(* CoDeSys 2.3 project: cy-wg-03_102.pro *)
(* Title: cy-003-wg (SanFelice) *)
(* Author: Andrea Ravasio *)
(* Libraries: serial_interface_01.lib 22.4.13 12:50:14, SerComm.lib 31.5.11 09:06:48, MBus_03.lib 9.2.13 17:51:58, Util.lib 26.9.14 11:12:46, Visual.lib 8.11.10 12:37:48, WagoLibIdent.lib 25.2.13 13:49:34, WagoLibStatus.lib 8.11.10 12:37:48, SysLibFile.lib 8.11.10 12:37:48, SysLibRtc.lib 8.11.10 12:37:48, SysLibSockets.lib 5.5.11 09:22:24, SysLibEvent.lib 8.11.10 12:37:48, SysLibPlcCtrl.lib 8.11.10 12:37:48, Standard.lib 8.11.10 12:37:48, SYSLIBCALLBACK.LIB 8.11.10 12:37:48, WagoLibDaylightSaving.lib 8.11.10 12:37:48, SysLibTime.lib 8.11.10 12:37:48, 32_Bit\DaylightSaving.lib 2.12.10 14:48:32 *)

(* PLC configuration (modules and I/O channels)
VPN_ST2 AT %IX16.0 [BOOLOnX_I] Ch_1 Digital input
KEY_QE_ST AT %IX16.1 [BOOLOnX_I] Ch_2 Digital input
SCA01_5_DI AT %IX16.2 [BOOLOnX_I] Ch_3 Digital input
PORT01_DI AT %IX16.3 [BOOLOnX_I] Ch_4 Digital input
0750-0402 4 DI 24 V DC 3.0ms [Type_1_4_Channels] node 1, in %IB32 out %QB8 {INTTypePAAssignment = PLC; INTTypeModule = plugged}
  GAS02_DI AT %IX16.4 [BOOLOnX_I] Ch_1 Digital input
  GAS01_DI AT %IX16.5 [BOOLOnX_I] Ch_2 Digital input
  SCA01_6_DI AT %IX16.6 [BOOLOnX_I] Ch_3 Digital input
  SCA05_1_DI AT %IX16.7 [BOOLOnX_I] Ch_4 Digital input
SCA05_2_DI AT %IX16.8 [BOOLOnX_I] Ch_1 Digital input
SCA01_1_DO AT %QX4.0 [BOOLOnX_Q] Ch_1 Digital output
SCA05_3_DI AT %IX16.9 [BOOLOnX_I] Ch_2 Digital input
SCA01_2_DO AT %QX4.1 [BOOLOnX_Q] Ch_2 Digital output
SCA05_4_DI AT %IX16.10 [BOOLOnX_I] Ch_3 Digital input
SCA01_3_DO AT %QX4.2 [BOOLOnX_Q] Ch_3 Digital output
SCA05_5_DI AT %IX16.11 [BOOLOnX_I] Ch_4 Digital input
SCA01_4_DO AT %QX4.3 [BOOLOnX_Q] Ch_4 Digital output
SCA05_6_DI AT %IX16.12 [BOOLOnX_I] Ch_5 Digital input
LAMP_AL AT %QX4.4 [BOOLOnX_Q] Ch_5 Digital output
AT %IX16.13 [BOOLOnX_I] Ch_6 Digital input
CAL02_RESET AT %QX4.5 [BOOLOnX_Q] Ch_6 Digital output
AT %IX16.14 [BOOLOnX_I] Ch_7 Digital input
CAL03_RESET AT %QX4.6 [BOOLOnX_Q] Ch_7 Digital output
SCA05_10_DI AT %IX16.15 [BOOLOnX_I] Ch_8 Digital input
AT %QX4.7 [BOOLOnX_Q] Ch_8 Digital output
SCA06_1_DI AT %IX17.0 [BOOLOnX_I] Ch_1 Digital input
CIRD02B_EN AT %QX4.8 [BOOLOnX_Q] Ch_1 Digital output
SCA06_2_DI AT %IX17.1 [BOOLOnX_I] Ch_2 Digital input
CIRD02A_EN AT %QX4.9 [BOOLOnX_Q] Ch_2 Digital output
SCA06_5_DI AT %IX17.2 [BOOLOnX_I] Ch_3 Digital input
CIRD01B_EN AT %QX4.10 [BOOLOnX_Q] Ch_3 Digital output
SCA06_6_DI AT %IX17.3 [BOOLOnX_I] Ch_4 Digital input
CIRD01A_EN AT %QX4.11 [BOOLOnX_Q] Ch_4 Digital output
SCA06_7_DI AT %IX17.4 [BOOLOnX_I] Ch_5 Digital input
EV02_EN AT %QX4.12 [BOOLOnX_Q] Ch_5 Digital output
SCA06_8_DI AT %IX17.5 [BOOLOnX_I] Ch_6 Digital input
EV03_EN AT %QX4.13 [BOOLOnX_Q] Ch_6 Digital output
SCA06_15_DI AT %IX17.6 [BOOLOnX_I] Ch_7 Digital input
CAL02_EN AT %QX4.14 [BOOLOnX_Q] Ch_7 Digital output
SCA06_16_DI AT %IX17.7 [BOOLOnX_I] Ch_8 Digital input
CAL03_EN AT %QX4.15 [BOOLOnX_Q] Ch_8 Digital output
0750-1506 8DI / 8DO 24V DC 0.5A [Type_34_8_Channels] node 4, in %IB34 out %QB9 {INTTypePAAssignment = PLC; INTTypeModule = plugged}
  SCA06_9_DI AT %IX17.8 [BOOLOnX_I] Ch_1 Digital input
  AT %QX5.0 [BOOLOnX_Q] Ch_1 Digital output
  SCA06_10_DI AT %IX17.9 [BOOLOnX_I] Ch_2 Digital input
  AT %QX5.1 [BOOLOnX_Q] Ch_2 Digital output
  SCA06_11_DI AT %IX17.10 [BOOLOnX_I] Ch_3 Digital input
  AT %QX5.2 [BOOLOnX_Q] Ch_3 Digital output
  SCA06_12_DI AT %IX17.11 [BOOLOnX_I] Ch_4 Digital input
  AT %QX5.3 [BOOLOnX_Q] Ch_4 Digital output
  SCA06_19_DI AT %IX17.12 [BOOLOnX_I] Ch_5 Digital input
  AT %QX5.4 [BOOLOnX_Q] Ch_5 Digital output
  SCA06_20_DI AT %IX17.13 [BOOLOnX_I] Ch_6 Digital input
  AT %QX5.5 [BOOLOnX_Q] Ch_6 Digital output
  CIRD01A_ST AT %IX17.14 [BOOLOnX_I] Ch_7 Digital input
  AT %QX5.6 [BOOLOnX_Q] Ch_7 Digital output
  CIRD01A_AL AT %IX17.15 [BOOLOnX_I] Ch_8 Digital input
  AT %QX5.7 [BOOLOnX_Q] Ch_8 Digital output
0750-1506 8DI / 8DO 24V DC 0.5A [Type_34_8_Channels] node 5, in %IB35 out %QB10 {INTTypePAAssignment = PLC; INTTypeModule = plugged}
  CIRD01B_ST AT %IX18.0 [BOOLOnX_I] Ch_1 Digital input
  AT %QX5.8 [BOOLOnX_Q] Ch_1 Digital output
  CIRD01B_AL AT %IX18.1 [BOOLOnX_I] Ch_2 Digital input
  AT %QX5.9 [BOOLOnX_Q] Ch_2 Digital output
  CIRD02A_ST AT %IX18.2 [BOOLOnX_I] Ch_3 Digital input
  AT %QX5.10 [BOOLOnX_Q] Ch_3 Digital output
  CIRD02A_AL AT %IX18.3 [BOOLOnX_I] Ch_4 Digital input
  AT %QX5.11 [BOOLOnX_Q] Ch_4 Digital output
  CIRD02B_ST AT %IX18.4 [BOOLOnX_I] Ch_5 Digital input
  AT %QX5.12 [BOOLOnX_Q] Ch_5 Digital output
  CIRD02B_AL AT %IX18.5 [BOOLOnX_I] Ch_6 Digital input
  AT %QX5.13 [BOOLOnX_Q] Ch_6 Digital output
  SCA04_1_DI AT %IX18.6 [BOOLOnX_I] Ch_7 Digital input
  TEST1 AT %QX5.14 [BOOLOnX_Q] Ch_7 Digital output
  SCA04_2_DI AT %IX18.7 [BOOLOnX_I] Ch_8 Digital input
  TEST2 AT %QX5.15 [BOOLOnX_Q] Ch_8 Digital output
0750-0430 8 DI 24 V DC 3.0ms [Type_1_8_Channels] node 6, in %IB36 out %QB11 {INTTypePAAssignment = PLC; INTTypeModule = plugged}
  SCA04_3_DI AT %IX18.8 [BOOLOnX_I] Ch_1 Digital input
  SCA04_7_DI AT %IX18.9 [BOOLOnX_I] Ch_2 Digital input
  SCA04_4_DI AT %IX18.10 [BOOLOnX_I] Ch_3 Digital input
  SCA04_8_DI AT %IX18.11 [BOOLOnX_I] Ch_4 Digital input
  SCA04_5_DI AT %IX18.12 [BOOLOnX_I] Ch_5 Digital input
  SCA04_9_DI AT %IX18.13 [BOOLOnX_I] Ch_6 Digital input
  SCA04_6_DI AT %IX18.14 [BOOLOnX_I] Ch_7 Digital input
  SCA04_10_DI AT %IX18.15 [BOOLOnX_I] Ch_8 Digital input
  SCA04_11_DI AT %IX19.0 [BOOLOnX_I] Ch_1 Digital input
  SCA05_9_DI AT %IX19.1 [BOOLOnX_I] Ch_2 Digital input
  SCA04_12_DI AT %IX19.2 [BOOLOnX_I] Ch_3 Digital input
  SCA05_11_DI AT %IX19.3 [BOOLOnX_I] Ch_4 Digital input
  SCA05_7_DI AT %IX19.4 [BOOLOnX_I] Ch_5 Digital input
  SCA05_12_DI AT %IX19.5 [BOOLOnX_I] Ch_6 Digital input
  SCA05_8_DI AT %IX19.6 [BOOLOnX_I] Ch_7 Digital input
  SCA04_13_DI AT %IX19.7 [BOOLOnX_I] Ch_8 Digital input
  SCA06_3_DI AT %IX19.8 [BOOLOnX_I] Ch_1 Digital input
  CIRD02B_AUTO AT %IX19.9 [BOOLOnX_I] Ch_2 Digital input
  SCA06_4_DI AT %IX19.10 [BOOLOnX_I] Ch_3 Digital input
  CIRD02A_AUTO AT %IX19.11 [BOOLOnX_I] Ch_4 Digital input
  SCA04_14_DI AT %IX19.12 [BOOLOnX_I] Ch_5 Digital input
  CIRD01B_AUTO AT %IX19.13 [BOOLOnX_I] Ch_6 Digital input
  SCA05_14_DI AT %IX19.14 [BOOLOnX_I] Ch_7 Digital input
  CIRD01A_AUTO AT %IX19.15 [BOOLOnX_I] Ch_8 Digital input
  SCA06_21_DI AT %IX20.0 [BOOLOnX_I] Ch_1 Digital input
  EV02_AUTO AT %IX20.1 [BOOLOnX_I] Ch_2 Digital input
  SCA06_22_DI AT %IX20.2 [BOOLOnX_I] Ch_3 Digital input
  EV03_OPEN AT %IX20.3 [BOOLOnX_I] Ch_4 Digital input
  EV02_OPEN AT %IX20.4 [BOOLOnX_I] Ch_5 Digital input
  EV03_CLOSE AT %IX20.5 [BOOLOnX_I] Ch_6 Digital input
  EV02_CLOSE AT %IX20.6 [BOOLOnX_I] Ch_7 Digital input
  EV03_AUTO AT %IX20.7 [BOOLOnX_I] Ch_8 Digital input
  SCA05_13_DI AT %IX20.8 [BOOLOnX_I] Ch_1 Digital input
  AT %IX20.9 [BOOLOnX_I] Ch_2 Digital input
  AT %IX20.10 [BOOLOnX_I] Ch_3 Digital input
  AT %IX20.11 [BOOLOnX_I] Ch_4 Digital input
  AT %IX20.12 [BOOLOnX_I] Ch_5 Digital input
  AT %IX20.13 [BOOLOnX_I] Ch_6 Digital input
  AT %IX20.14 [BOOLOnX_I] Ch_7 Digital input
  AT %IX20.15 [BOOLOnX_I] Ch_8 Digital input
0750-0430 8 DI 24 V DC 3.0ms [Type_1_8_Channels] node 11, in %IB41 out %QB12 {INTTypePAAssignment = PLC; INTTypeModule = plugged}
  AT %IX21.0 [BOOLOnX_I] Ch_1 Digital input
  AT %IX21.1 [BOOLOnX_I] Ch_2 Digital input
  AT %IX21.2 [BOOLOnX_I] Ch_3 Digital input
  AT %IX21.3 [BOOLOnX_I] Ch_4 Digital input
  AT %IX21.4 [BOOLOnX_I] Ch_5 Digital input
  AT %IX21.5 [BOOLOnX_I] Ch_6 Digital input
  AT %IX21.6 [BOOLOnX_I] Ch_7 Digital input
  AT %IX21.7 [BOOLOnX_I] Ch_8 Digital input
0750-0464#02 2/4 AI RTD / ADJ./ HA [Type_44_2_Channels] node 12, in %IB28 out %QB4 {INTTypePAAssignment = PLC; INTTypeModule = plugged}
  TT_S01 AT %IW0 [INTOnW_I] Ch_1 signed Input value
  AT %IW1 [INTOnW_I] Ch_2 signed Input value
0750-0472 2 AI 0-20mA 16 Bit S.E. [Type_8_2_Channels] node 13, in %IB28 out %QB4 {INTTypePAAssignment = PLC; INTTypeModule = plugged}
  TT_S07 AT %IW2 [WORDOnW_I] I 1: Analog Input
  TT_S06 AT %IW3 [WORDOnW_I] I 2: Analog Input
0750-0472 2 AI 0-20mA 16 Bit S.E. [Type_8_2_Channels] node 14, in %IB32 out %QB4 {INTTypePAAssignment = PLC; INTTypeModule = plugged}
  TT_S05 AT %IW4 [WORDOnW_I] I 1: Analog Input
  TT_S04 AT %IW5 [WORDOnW_I] I 2: Analog Input
0750-0472 2 AI 0-20mA 16 Bit S.E. [Type_8_2_Channels] node 15, in %IB36 out %QB4 {INTTypePAAssignment = PLC; INTTypeModule = plugged}
  TT_S03 AT %IW6 [WORDOnW_I] I 1: Analog Input
  TT_S02 AT %IW7 [WORDOnW_I] I 2: Analog Input
  PORT01_AI AT %IW8 [WORDOnW_I] I 1: Analog Input
  AT %IW9 [WORDOnW_I] I 2: Analog Input
  CAL02_ST_POTENZA AT %IW10 [WORDOnW_I] Ch_1 Input word
  CAL03_ST_POTENZA AT %IW11 [WORDOnW_I] Ch_2 Input word
0750-0472 2 AI 0-20mA 16 Bit S.E. [Type_8_2_Channels] node 18, in %IB48 out %QB4 {INTTypePAAssignment = PLC; INTTypeModule = plugged}
  TT_S09 AT %IW12 [WORDOnW_I] Ch_1 Input word
  TT_S08 AT %IW13 [WORDOnW_I] Ch_2 Input word
0750-0556 2 AO ±10V [Type_14_2_Channels] node 19, in %IB52 out %QB4 {INTTypePAAssignment = PLC; INTTypeModule = plugged}
  CAL02_SETPOINT AT %QW0 [WORDOnW_Q] Ch_1 Analog output
  CAL03_SETPOINT AT %QW1 [WORDOnW_Q] Ch_2 Analog output
0750-0650/0003-0000#03 RS 232 C Interface (Adjustable), 3 Byte [Type_21_1_Channels] node 20, in %IB56 out %QB4 {INTTypePAAssignment = PLC; INTTypeModule = plugged}
  AT %IX14.0 [BOOLOnX_I] Transmission acknowledgement
  AT %IX14.1 [BOOLOnX_I] Reception request
  AT %IX14.2 [BOOLOnX_I] Initialization acknowledgement
  AT %IX14.3 [BOOLOnX_I] Input buffer is full
  AT %IX14.4 [BOOLOnX_I] Number of received characters Bit 0
  AT %IX14.5 [BOOLOnX_I] Number of received characters Bit 1
  AT %IX14.6 [BOOLOnX_I] Number of received characters Bit 2
  AT %IB29 [BYTEOnB_I] Input data Byte 0
  AT %IB30 [BYTEOnB_I] Input data Byte 1
  AT %IB31 [BYTEOnB_I] Input data Byte 2
  AT %QX2.0 [BOOLOnX_Q] Transmission request
  AT %QX2.1 [BOOLOnX_Q] Reception acknowledgement
  AT %QX2.2 [BOOLOnX_Q] Initialization request
  AT %QX2.4 [BOOLOnX_Q] Number of characters Bit 0
  AT %QX2.5 [BOOLOnX_Q] Number of characters Bit 1
  AT %QX2.6 [BOOLOnX_Q] Number of characters Bit 2
  AT %QB5 [BYTEOnB_Q] Output data Byte 0
  AT %QB6 [BYTEOnB_Q] Output data Byte 1
  AT %QB7 [BYTEOnB_Q] Output data Byte 2
Fieldbus variables [FB_VARS] node 1, in %IB0 out %QB0
Flag variables [FLAG_VARS] node 2, in %IB0 out %QB0
Modbus-Master [MB_MASTER] node 3, in %IB0 out %QB0
*)

(* Task configuration *)
TASK FastCounter (PRIORITY := 5, INTERVAL := T#3ms);
	PLC_FAST_CTR();
END_TASK
TASK Main (PRIORITY := 10); (* freewheeling *)
	PLC_PRG();
END_TASK
TASK ConteggioGas1 (PRIORITY := 2, SINGLE := GAS01_DI);
	ConteggioGAS1();
END_TASK
TASK ConteggioGAS2 (PRIORITY := 1, SINGLE := GAS02_DI);
	ConteggioGAS2();
END_TASK

(* Global variable list: Global_Constants *)
VAR_GLOBAL CONSTANT

	Plant_NAME			: STRING :='cySN:3 cyVER:100 - San Felice';
	Plant_SN			: DWORD :=3;   		(* S/N Impianto di telecontrollo *)
	Plant_SW_VER		: WORD  :=100;		(* Versione SW installata *)

	(* Parameters *)
	Plant_DefaultTAmb	: INT	:=-9999;	(* [.1°C] Temperatura ambiente di default in caso di rottura sonda *)

	(* Filesystem *)
	FilesPath  			: STRING :='S:\';

	(* TCP Logger *)
	Logger_SERVER		: STRING:='';
	Logger_IP			: STRING:='192.168.100.3';
	Logger_PORT			: WORD  :=80;
	Logger_GETSTART		: STRING:='GET /cygmsrv/hsgm.ashx?';
	Logger_GETEND		: STRING:='$R$N$R$N';
	Logger_CHECK		: STRING:='True';
	Logger_CRLF			: STRING:='$R$N';
	Logger_DataFile		: STRING:='S:\LOG.DAT';
	Logger_DataFileOld	: STRING:='S:\LOG.BCK';
	Logger_IndexFile	: STRING:='S:\LOG1.IDX';
	Logger_ConnRetries	: BYTE:=5;
	Logger_RecoverMsgs	: BYTE:=100;

	(* TCP Remote *)
	Remote_PORT			: WORD  :=10;
	Remote_WELCOME		: STRING:='Connected$R$N';
	Remote_OK			: STRING:='OK$R$N';
	Remote_ERROR		: STRING:='ERROR$R$N';

	(* TCP Sockets *)
	MAX_SEND_TCP_SERVER					 : DWORD:=1500;(*60000*)
	MAX_RECEIVE_TCP_SERVER				 : DWORD:=3000;
	MAX_RECEIVE_TCP_SERVER_SOCKET	 	 : DWORD:=1500;
	MAX_SEND_TCP_CLIENT					 : DWORD:=3000;(*15000*)
	MAX_RECEIVE_TCP_CLIENT				 : DWORD:=1500;
	MAX_RECEIVE_TCP_CLIENT_SOCKET		 : DWORD:=1500;
	MAX_RECEIVE_UDP_SERVER				 : INT  :=1472;
	MAX_RECEIVE_UDP_CLIENT				 : INT  :=1472;
	CONNECT_WATCHDOG_TIME				 : TIME :=t#10s;

	(* VISU COLORS *)
	COLOR_RED 			: DWORD:=16#2020F0;
	COLOR_YELLOW		: DWORD:=16#20F0F0;
	COLOR_GREEN			: DWORD:=16#20F020;
	COLOR_GREEN_OFF 	: DWORD:=16#006000;
	COLOR_LBLUE			: DWORD:=16#F0F080;
	COLOR_GREY			: DWORD:=16#C0C0C0;

END_VAR
VAR_GLOBAL
	ChangeGAS1: BOOL;
	OffsetContatoreGAS1_1W: DINT;
	OffsetContatoreGAS1_2W: DINT;
	OffsetGAS1: DINT;

	ChangeGAS2: BOOL;
	OffsetContatoreGAS2_1W: DINT;
	OffsetContatoreGAS2_2W: DINT;
	OffsetGAS2: DINT;

END_VAR

(* Global variable list: Global_Retain *)
VAR_GLOBAL RETAIN PERSISTENT

	PortataTotalePORT01		: DINT;
	ConteggioTotalePORT01	: DINT;
	PortataTotaleGAS01		: DINT;
	ConteggioTotaleGAS01	: DINT;
	PortataTotaleGAS02		: DINT;
	ConteggioTotaleGAS02	: DINT;

	CTB250_ENERGY_WH		: REAL;
	CTB250_ENERGY			: DWORD; (* 10^-2 MWh *)

	Mode_Manual : BOOL := FALSE;

	CAL02_Clima : typ_Clima;
	CAL03_Clima : typ_Clima;

	DelayAllarmeTemperaturaNonRaggiunta: INT;
	DeltaInterventoAllarmeTempeaturaNonRaggiuta: INT;
	OffsetSetPointManuale:INT;							(* Offset al Setpoint manuale per comensare lo scambiatore *)




END_VAR

(* Global variable list: Global_Variables *)
VAR_GLOBAL

	SYS    : typ_SYS;
	T_AMB  : INT;

	TPV01  : obj_TPV		:= ( ID:=1,
								 IN_EMIN:=-600 , IN_EMAX:=2500 ,
								 IN_WMIN:=-500 , IN_WMAX:=600 ); (* T_S01 *)

	TPV02  : obj_TPV_SENS	:= ( ID:=2 ,
											SogliaHL:=4096 ,   	 	(* Soglia Sonda Aperta = 2,5mA *)
											SogliaHH:=32767,	 	(* Soglia Sonda CC = 20mA *)
											SogliaWL:=10, 			(* Soglia WRN Bassa  = 10°C *)
											SogliaWH:=120,			(* Soglia WRN Alta  = 120°C *)
											PuntoMinX:=0, 		    (* Scalatura Minima vedi data di targa sonda 0°C *)
											PuntoMaxX:=160,			(* Scalatura Massima Vedi data di targa Sonda 160°C *)
											PuntoMinY:=6553,		(* Valore minimio per scalatura = 4mA *)
											PuntoMaxY:=32767,		(* Valore Massimo per Scalatura = 20mA *)
											Decimali:=1); 			(* Decimali da ottenere durante la scalatura *)
	TPV03  : obj_TPV_SENS	:= ( ID:=3 ,
											SogliaHL:=4096 ,   	 	(* Soglia Sonda Aperta = 2,5mA *)
											SogliaHH:=32767,	 	(* Soglia Sonda CC = 20mA *)
											SogliaWL:=10, 			(* Soglia WRN Bassa  = 10°C *)
											SogliaWH:=120,			(* Soglia WRN Alta  = 120°C *)
											PuntoMinX:=0, 		    (* Scalatura Minima vedi data di targa sonda 0°C *)
											PuntoMaxX:=160,			(* Scalatura Massima Vedi data di targa Sonda 160°C *)
											PuntoMinY:=6553,		(* Valore minimio per scalatura = 4mA *)
											PuntoMaxY:=32767,		(* Valore Massimo per Scalatura = 20mA *)
											Decimali:=1); 			(* Decimali da ottenere durante la scalatura *)

	TPV04  : obj_TPV_SENS	:= ( ID:=4 ,
											SogliaHL:=4096 ,   	 	(* Soglia Sonda Aperta = 2,5mA *)
											SogliaHH:=32767,	 	(* Soglia Sonda CC = 20mA *)
											SogliaWL:=10, 			(* Soglia WRN Bassa  = 10°C *)
											SogliaWH:=120,			(* Soglia WRN Alta  = 120°C *)
											PuntoMinX:=0, 		    (* Scalatura Minima vedi data di targa sonda 0°C *)
											PuntoMaxX:=160,			(* Scalatura Massima Vedi data di targa Sonda 160°C *)
											PuntoMinY:=6553,		(* Valore minimio per scalatura = 4mA *)
											PuntoMaxY:=32767,		(* Valore Massimo per Scalatura = 20mA *)
											Decimali:=1); 			(* Decimali da ottenere durante la scalatura *)

	TPV05  : obj_TPV_SENS	:= ( ID:=5 ,
											SogliaHL:=4096 ,   	 	(* Soglia Sonda Aperta = 2,5mA *)
											SogliaHH:=32767,	 	(* Soglia Sonda CC = 20mA *)
											SogliaWL:=10, 			(* Soglia WRN Bassa  = 10°C *)
											SogliaWH:=120,			(* Soglia WRN Alta  = 120°C *)
											PuntoMinX:=0, 		    (* Scalatura Minima vedi data di targa sonda 0°C *)
											PuntoMaxX:=160,			(* Scalatura Massima Vedi data di targa Sonda 160°C *)
											PuntoMinY:=6553,		(* Valore minimio per scalatura = 4mA *)
											PuntoMaxY:=32767,		(* Valore Massimo per Scalatura = 20mA *)
											Decimali:=1); 			(* Decimali da ottenere durante la scalatura *)

	TPV06  : obj_TPV_SENS	:= ( ID:=6 ,
											SogliaHL:=4096 ,   	 	(* Soglia Sonda Aperta = 2,5mA *)
											SogliaHH:=32767,	 	(* Soglia Sonda CC = 20mA *)
											SogliaWL:=10, 			(* Soglia WRN Bassa  = 10°C *)
											SogliaWH:=120,			(* Soglia WRN Alta  = 120°C *)
											PuntoMinX:=0, 		    (* Scalatura Minima vedi data di targa sonda 0°C *)
											PuntoMaxX:=160,			(* Scalatura Massima Vedi data di targa Sonda 160°C *)
											PuntoMinY:=6553,		(* Valore minimio per scalatura = 4mA *)
											PuntoMaxY:=32767,		(* Valore Massimo per Scalatura = 20mA *)
											Decimali:=1); 			(* Decimali da ottenere durante la scalatura *)

	TPV07  : obj_TPV_SENS	:= ( ID:=7 ,
											SogliaHL:=4096 ,   	 	(* Soglia Sonda Aperta = 2,5mA *)
											SogliaHH:=32767,	 	(* Soglia Sonda CC = 20mA *)
											SogliaWL:=10, 			(* Soglia WRN Bassa  = 10°C *)
											SogliaWH:=120,			(* Soglia WRN Alta  = 120°C *)
											PuntoMinX:=0, 		    (* Scalatura Minima vedi data di targa sonda 0°C *)
											PuntoMaxX:=160,			(* Scalatura Massima Vedi data di targa Sonda 160°C *)
											PuntoMinY:=6553,		(* Valore minimio per scalatura = 4mA *)
											PuntoMaxY:=32767,		(* Valore Massimo per Scalatura = 20mA *)
											Decimali:=1); 			(* Decimali da ottenere durante la scalatura *)

	TPV08  : obj_TPV_SENS	:= ( ID:=8 ,
											SogliaHL:=4096 ,   	 	(* Soglia Sonda Aperta = 2,5mA *)
											SogliaHH:=32767,	 	(* Soglia Sonda CC = 20mA *)
											SogliaWL:=10, 			(* Soglia WRN Bassa  = 10°C *)
											SogliaWH:=120,			(* Soglia WRN Alta  = 120°C *)
											PuntoMinX:=0, 		    (* Scalatura Minima vedi data di targa sonda 0°C *)
											PuntoMaxX:=160,			(* Scalatura Massima Vedi data di targa Sonda 160°C *)
											PuntoMinY:=6553,		(* Valore minimio per scalatura = 4mA *)
											PuntoMaxY:=32767,		(* Valore Massimo per Scalatura = 20mA *)
											Decimali:=1); 			(* Decimali da ottenere durante la scalatura *)
	TPV09  : obj_TPV_SENS	:= ( ID:=9 ,
											SogliaHL:=4096 ,   	 	(* Soglia Sonda Aperta = 2,5mA *)
											SogliaHH:=32767,	 	(* Soglia Sonda CC = 20mA *)
											SogliaWL:=10, 			(* Soglia WRN Bassa  = 10°C *)
											SogliaWH:=120,			(* Soglia WRN Alta  = 120°C *)
											PuntoMinX:=0, 		    (* Scalatura Minima vedi data di targa sonda 0°C *)
											PuntoMaxX:=160,			(* Scalatura Massima Vedi data di targa Sonda 160°C *)
											PuntoMinY:=6553,		(* Valore minimio per scalatura = 4mA *)
											PuntoMaxY:=32767,		(* Valore Massimo per Scalatura = 20mA *)
											Decimali:=1); 			(* Decimali da ottenere durante la scalatura *)

	(* Misuratore di Portata *)
	PORT01  : obj_PORT	:=  ( ID:=1 ,
											TempoTimeOut:=T#2m,		(* PULSE - Minuti di attesa prima di segnalare WRN di inattività sulla linea *)
											SogliaHL:=4096,   	 	(* FLOW - Soglia Sonda Aperta = 2,5mA *)
											SogliaHH:=32767,	 	(* FLOW - Soglia Sonda CC = 20mA *)
											SogliaWL:=100000, 		(* FLOW - [E-3 m3/h] Soglia WRN Bassa *)
											SogliaWH:=700000,		(* FLOW - [E-3 m3/h] Soglia WRN Alta *)
											PuntoMinX:=0, 		    (* FLOW - [E-3 m3/h] Scalatura minima vedi data di targa sonda *)
											PuntoMaxX:=800000,		(* FLOW - [E-3 m3/h] Scalatura massima Vedi data di targa sonda *)
											PuntoMinY:=6553,		(* FLOW - Valore minimio per scalatura = 4mA *)
											PuntoMaxY:=32767		(* FLOW - Valore massimo per Scalatura = 20mA *)
											);

	(*  Contatori *)
	GAS01  : obj_GAS:=  (ID:=1,	Peso:=1 ,				(* Peso del'impulso *)
								TempoTimeOut:=T#15m		(* Minuti di attesa prima di segnalare WRN di inattività sulla linea *)
													  );
	GAS02  : obj_GAS:=  (ID:=2,	Peso:=1 ,				(* Peso del'impulso *)
								TempoTimeOut:=T#15m		(* Minuti di attesa prima di segnalare WRN di inattività sulla linea *)
													  );


	CronEd	: 	obj_CRON_EDITOR;

	(* CRONOTERMOSTATI *)
	THER01 : obj_CRONTER := ( ID:=1, Local_MaxRunTAmb:=900,Histeresys:=10); (* Controllo CIRD01 *)
	THER02 : obj_CRONTER := ( ID:=2, Local_MaxRunTAmb:=900,Histeresys:=10);	(* Controllo CIRD02 *)
	THER03 : obj_CRONTER := ( ID:=3, Local_MaxRunTAmb:=900,Histeresys:=10);	(* Controllo CAL02 *)
	THER04 : obj_CRONTER := ( ID:=4, Local_MaxRunTAmb:=900,Histeresys:=10);	(* Controllo CAL03 *)

	(* Circolatori  *)
	CIRD01 :obj_CIRD_01 := (ID:=1, OnDelay:=T#10ms,OffDelay:=T#10ms, Mode:=3); (* Circolatore P2 scorta - P3 prioritario *)
	CIRD02 :obj_CIRD_01 := (ID:=2, OnDelay:=T#10ms,OffDelay:=T#10ms, Mode:=2); (* Circolatore P4 prioritario - P5 scorta *)

	(* Elettrovalvole  *) (* con Mod_ComandoEV=0 la valvola è NA con comando a 1 si apre,con Mod_ComandoEV=1	la valvola è NC con comando a 1 si chiude  *)
	EV02 :obj_EV_01 := (ID:=2, OnDelay:=T#1s,OffDelay:=T#15m, Mod_ComandoEV:=FALSE); (* EV02 su CAL02 *)
	EV03 :obj_EV_01 := (ID:=3, OnDelay:=T#1s,OffDelay:=T#15m, Mod_ComandoEV:=FALSE); (* EV03 su CAL03 *)

	(* Caldaie *)
	CAL02  : obj_CAL_01 := ( ID:=2,	LimiteMAXSetPoint:= 1400,LimiteMinSetPoint:=600,OnDelay:=T#10m,OffDelay:=T#500ms );
	CAL03  : obj_CAL_01 := ( ID:=3,	LimiteMAXSetPoint:= 1400,LimiteMinSetPoint:=600,OnDelay:=T#10m,OffDelay:=T#500ms );





	(* MBUS Contabilizers *)
	MBUS01 	  : obj_MBUS				:= ( ID:=1 , COM:=2 , BAUDRATE:=BAUD_2400 );
	CTBSCAN01 : obj_MBUS_CTB_SCANNER	:= ( ID:=1 );
	(*---- MBUS DEBUG ----*)
(*	COMx					: SERIAL_INTERFACE := (bCOM_PORT_NR		:= 2,
			cbBAUDRATE			:= BAUD_2400,
			cbsBYTESIZE			:= BS_8,
			cpPARITY			:= PARITY_EVEN,
			csSTOPBITS			:= STOPBITS_1,
			cfFLOW_CONTROL		:= NO_FLOW_CONTROL);
	RXBuf					: typRING_BUFFER;
	TXBuf					: ARRAY [0..16] OF BYTE;
	xINI					: BOOL;
	xSND					: BOOL;
	maddress : BYTE;
	mchk : BYTE;
	mt1 : BOOL;
	mt2 : BOOL;
	mt3 : BOOL;
*)

	(* Virtual contabilizers *)
	CTB250	  : obj_SW_CTB				:= ( ID:=250 );

	Logger : typ_Logger;



	(* Gestione ora solare , giorno *)

	OraLegale: BOOL;
	NomeGiorno:BYTE;


	(**** SIMULATION ONLY ****)
	(*...*)
END_VAR

(* Data type in Errors *)
TYPE en_Logger_ErrLev :
(
	EL_Log			:=0,
	EL_Wrn			:=1,
	EL_Alarm		:=2,
	EL_AlarmStop	:=3
);
END_TYPE

(* Data type in Errors *)
TYPE en_Logger_Status :
(
	S_Logger_UNKNOWN := 0,
	S_Logger_IDLE,
	S_Logger_WAITCONN,
	S_Logger_WAITTX,
	S_Logger_WAITRESP,
	S_Logger_ERROR
);
END_TYPE

(* Data type *)
TYPE en_SYS_Objects :
(
	EO_SYS		:=0,  (* PLC *)
	EO_VPN		:=1,  (* VPN *)
	EO_DOOR		:=2,  (* Door & access control *)

	EO_CAL		:=10, (* Caldaia *)
	EO_CIR		:=11, (* Circolatore *)
	EO_CRON		:=12, (* Crono-termostato *)
	EO_VRD		:=13, (* Valvola miscelatore pannelli *)
	EO_CTL		:=14, (* Contalitri *)
	EO_CTB		:=15, (* Contabilizzatore *)
	EO_TPV		:=16, (* Temperature probes values *)
	EO_PPV		:=17, (* Pressure probes values *)
	EO_PBV		:=18, (* Over-Pressure Alarms *)
	EO_TBV		:=19, (* Over-Temperature Alarms *)
	EO_PMV		:=20, (* Under-Pressure Alarms *)
	EO_GRU		:=21, (* Gruppo termico *)
	EO_PDC		:=22, (* Pompa di calore *)
	EO_SOL		:=23, (* Pannello solare termico *)
	EO_ESOL		:=24, (* Pannello solare fotovoltaico *)
	EO_GAS		:=25, (* Contatore GAS *)
	EO_PORT		:=26, (* Misuratore di portata *)
	EO_FPV		:=27, (* Flow probes values *)
	EO_ANZ		:=28, (* Analizzatore di rete *)
	EO_SCA		:=29, (* Signal Control Alarms *)
	EO_LUX		:=30, (* Base Illumination point *)
	EO_LUXM		:=31, (* Metered Illumination point *)
	EO_PSG		:=32, (* Sensore di passaggio *)
	EO_HVAC		:=33, (* Heating, Ventilating and Air Conditioning *)
	EO_HYGRV	:=34, (* Relative Humidity sensors value *)
	EO_COOV		:=35, (* Carbon Dioxide CO2 sensors value *)
	EO_INV		:=36, (* Inverter *)
	EO_STR		:=37, (* Smart string box *)

	EO_SPT		:=38, (* SPLIT *)

	EO_CIRD		:=39, (* Double CIR *)
	EO_ACS		:=40, (* Hot domestic water *)
	EO_FRG		:=41, (* Frigo *)
	EO_THER		:=42, (* Thermostat *)
	EO_CIRM		:=43, (* Modbus CIR *)
	EO_CIRDM	:=44, (* Modbus double CIR *)

	EO_EV		:=45, (* Elettrovalvole *)


	EO_ZGW			:=200,  (* ZigBee - Gateway *)
	EO_ZRM			:=201,	(* ZigBee - Repeater *)
	EO_ZREL			:=202,	(* ZigBee - Actuator rele *)
	EO_ZTHL			:=203,	(* ZigBee - Temperature Sensor *)

	EO_ASGW			:=250,	(* ASi - Gateway *)
	EO_ASCBI		:=251,	(* ASi - Input Board, Ciabatta *)

	EO_LON			:=1000, (* Bus - LON *)
	EO_MODBUS		:=1001, (* Bus - MODBUS *)
	EO_MBUS			:=1002, (* Bus - M-BUS *)
	EO_MODBUS_TCP	:=1003, (* Bus - MODBUS TCP *)

	EO_GENERIC		:=9000, (* Generic dataset *)
	EO_EXPO			:=9001 (* EXPO dataset *)

);
END_TYPE

(* Data type *)
TYPE en_SYS_Status :
(
	S_UNKNOWN  := 0,
	S_STARTUP,
	S_INIT_RTC,
	S_INIT_VAR,
	S_AUTOTEST,
	S_RUNNING,
	S_SHUTDOWN,
	S_HALT
);
END_TYPE

(* Data type in Plant_Objects *)
TYPE typ_Clima : (* CURVA CLIMATICA *)
STRUCT
	InitOK:		BOOL;
	Points: 	ARRAY [0..10] OF POINT;
END_STRUCT
END_TYPE

(* Data type in Plant_Objects *)
TYPE typ_Cron_Calendar :
STRUCT
	Profile		: ARRAY[0..384] OF BYTE;
END_STRUCT
END_TYPE

(* Data type in Plant_Objects *)
TYPE typ_Cron_Jolly :
STRUCT
	Start		: DT;
	End			: DT;
	Temp		: WORD;
	Flags		: WORD; (* B0:Enabled B1..B15:Unused *)
END_STRUCT
END_TYPE

(* Data type in Plant_Objects *)
TYPE typ_Cron_Profile :
STRUCT
	Flags		: WORD;
	Setpoint	: ARRAY [0..95] OF WORD;
END_STRUCT
END_TYPE

(* Data type in Errors *)
TYPE typ_Logger :
STRUCT
	Status		: en_Logger_Status;

	SendReq		: BOOL;
	SendIdx		: DWORD;
	SendData	: ARRAY [0..MAX_SEND_TCP_CLIENT] OF BYTE;
	SendLen		: DINT;

	TData		: ARRAY [0..MAX_SEND_TCP_CLIENT] OF BYTE;
	TLen		: DINT;

	LastIdxPos	: DWORD;

	(* Temporary variables used by objects *)
	s1			: STRING(256);
	i1			: WORD;

END_STRUCT
END_TYPE

(* Data type in Plant_Objects *)
TYPE typ_MBUS_CTBS :
STRUCT
	Present			: BOOL;
	Address			: DWORD;
	NodeError		: BYTE;

	Info			: typMBusInfo;
	Data_FTemp	 	: REAL; (* C *)
	Data_RTemp	 	: REAL; (* C *)
	Data_Flow	 	: REAL; (* m3ph *)
	Data_Power	 	: REAL; (* W *)
	Data_Energy 	: REAL; (* kWh *)

	Status_Log		: BYTE;
	Status_Vis		: DWORD;

END_STRUCT
END_TYPE

(* Data type *)
TYPE typ_SYS :
STRUCT
	Status			: en_SYS_Status;
	Warning			: BOOL;
	Alarm			: BOOL;
	AlarmStop		: BOOL;

	Time_LogString	: STRING;
	Time_Year		: WORD;
	Time_Month		: BYTE;
	Time_Day		: BYTE;

	Time_CT_DT		: DT;
	Time_CT_Day		: WORD;
	Time_CT_Quarter	: BYTE;

	LastLogs_Idx	: BYTE;
	LastLogs_Dat	: ARRAY[0..5] OF STRING;
	LastLogs_Msg	: ARRAY[0..5] OF STRING;

END_STRUCT
END_TYPE

(* Data type in Plant_Objects *)
TYPE typ_VisuStrutturaMbus :
STRUCT

	sdNodoPresente: STRING(16);
	sdEnergia: STRING(16);
	sdPotenza: STRING(16);
	sdVolume: STRING(16);
	sdFlow: STRING(16);
	sdTempIngresso: STRING(8);
	sdTempaUscita: STRING(8);
	sdTempDelta: STRING(8);

END_STRUCT
END_TYPE

(* POU PLC_FAST_CTR, ST *)
PROGRAM PLC_FAST_CTR
VAR
END_VAR
GAS01.Count(Contatore:=ConteggioTotaleGAS01, Totalizzatore:=PortataTotaleGAS01);
GAS02.Count(Contatore:=ConteggioTotaleGAS02, Totalizzatore:=PortataTotaleGAS02);
END_PROGRAM

(* POU PLC_PRG, ST *)
PROGRAM PLC_PRG
VAR
	Timer1: TON; (* Fast controls tick *)
	Timer2: TON; (* Plant control tick *)
	Timer3: TON; (* Logger timer *)

	t_sum : INT; (* Vars for dynamic means of working probes *)
	t_cnt : INT;
	CIRD03: BOOL;
	SendLog: BOOL;
	delFileIdx: BOOL;
	DelayOffPompe: TOF;
END_VAR
(******************************************************************************
 ****                           MAIN TASK CODE                             ****
 ******************************************************************************

	Network setup:
		IP  = 192.168.100.2 | MSK = 255.255.255.0 | GW = 192.168.100.1
		DNS = 192.168.100.1 | NTP = 193.168.100.3

	Editor setup:
		Project --> Options --> Editor --> Fonts --> Courier NEW / BOLD / 12

*)

(*==============================*)
(*===== Main status machine ====*)
(*==============================*)
Main_Stm();

(*=====================================*)
(*== Running common cycle operations ==*)
(*=====================================*)
IF SYS.Status>S_INIT_VAR THEN

	(* Execute M-BUS processes *)
	MBUS01();
	CTBSCAN01( MBUS:=MBUS01 );

	GAS01 ( GAS_DI:=GAS01_DI, Totalizzatore:=PortataTotaleGAS01, Contatore:=ConteggioTotaleGAS01 );
	GAS02 ( GAS_DI:=GAS02_DI, Totalizzatore:=PortataTotaleGAS02, Contatore:=ConteggioTotaleGAS02 );


			CIRD01(
					PumpA_AUTO:= CIRD01A_AUTO,
					PumpB_AUTO:= CIRD01b_AUTO ,
				(*	PumpA_En=>CIRD01a_EN ,
					PumpB_EN=>CIRD01b_EN , *)
					PumpA_AL:=NOT CIRD01A_AL,
					PumpB_AL:=NOT CIRD01B_AL,
					PumpA_ST:=CIRD01a_ST ,
					PumpB_ST:=CIRD01b_ST );

				(* introduzione di questa sicuurezza per evitare che le pompe partano senza avere lo sfogo *)
					CIRD01a_EN:=CIRD01.PumpA_En AND (EV02.EV_Open OR EV03.EV_Open);
					CIRD01b_EN:=CIRD01.PumpB_En AND (EV02.EV_Open OR EV03.EV_Open);




			CIRD02(
					PumpA_AUTO:= CIRD02a_AUTO,
					PumpB_AUTO:= CIRD02b_AUTO,
				(*	PumpA_En=>CIRD02a_EN ,
					PumpB_EN=>CIRD02b_EN , *)
					PumpA_AL:=NOT CIRD02a_AL,
					PumpB_AL:=NOT CIRD02b_AL,
					PumpA_ST:=CIRD02a_ST ,
					PumpB_ST:=CIRD02b_ST );


				(* introduzione di questa sicuurezza per evitare che le pompe partano senza avere lo sfogo *)
					CIRD02a_EN:=CIRD02.PumpA_En AND (EV02.EV_Open OR EV03.EV_Open);
					CIRD02b_EN:=CIRD02.PumpB_En AND (EV02.EV_Open OR EV03.EV_Open);




			EV02( 	EV_Open:= EV02_OPEN,
					EV_Close:=EV02_CLOSE ,
					EV_Auto:=EV02_AUTO ,
					EV_En=>EV02_EN ,
	 				);

			EV03( 	EV_Open:= EV03_OPEN,
					EV_Close:=EV03_CLOSE ,
					EV_Auto:=EV03_AUTO ,
					EV_En=>EV03_EN ,
	 				);

 			CAL02(AI_Potenza:= CAL02_ST_POTENZA,
					CAL_ST:=SCA_Proc.SCA04_2.OUT,
					ALARM_CAL:= SCA_Proc.SCA04_1.OUT OR
								SCA_Proc.SCA04_3.OUT OR
								SCA_Proc.SCA04_4.OUT OR
								SCA_Proc.SCA04_5.OUT OR
								SCA_Proc.SCA04_6.OUT OR
								SCA_Proc.SCA04_7.OUT OR
								SCA_Proc.SCA04_8.OUT OR
								SCA_Proc.SCA04_9.OUT OR
								SCA_Proc.SCA04_10.OUT OR
								SCA_Proc.SCA04_11.OUT(*	 OR
								SCA_Proc.SCA04_12.OUT OR
								SCA_Proc.SCA04_13.OUT *) ,
					PresenzaFiamma:=SCA_Proc.SCA04_2.OUT,
					CmdCALAuto_MAN:= SCA_Proc.SCA04_12.OUT,
					CLIM:=CAL02_Clima ,
					AO_SetPoint=>CAL02_SETPOINT ,
					CAL_EN=>CAL02_EN ,
					DO_RIARMO=>CAL02_RESET ,
					 );

 			CAL03(AI_Potenza:= CAL03_ST_POTENZA,
					CAL_ST:=SCA_Proc.SCA05_2.OUT,
					ALARM_CAL:= SCA_Proc.SCA05_1.OUT OR
								SCA_Proc.SCA05_3.OUT OR
								SCA_Proc.SCA05_4.OUT OR
								SCA_Proc.SCA05_5.OUT OR
								SCA_Proc.SCA05_6.OUT OR
								SCA_Proc.SCA05_7.OUT OR
								SCA_Proc.SCA05_8.OUT OR
								SCA_Proc.SCA05_9.OUT OR
								SCA_Proc.SCA05_10.OUT OR
								SCA_Proc.SCA05_11.OUT (*OR
								SCA_Proc.SCA05_12.OUT OR
								SCA_Proc.SCA05_13.OUT *) ,
					PresenzaFiamma:=SCA_Proc.SCA05_2.OUT,
					CmdCALAuto_MAN:= SCA_Proc.SCA05_12.OUT,
					CLIM:=CAL03_Clima ,
					AO_SetPoint=>CAL03_SETPOINT ,
					CAL_EN=>CAL03_EN ,
					DO_RIARMO=>CAL03_RESET ,
					 );






(* Lamp.UpdateStatus(obj_Status := Status_Log); *)



(*	COMx(	ptSEND_BUFFER		:= ADR(TXBuf),
			xSTART_SEND			:= xSND,
			utRECEIVE_BUFFER	:= RXBuf,
			xINIT				:= xINI );

	IF mt1 THEN
		mt1:=FALSE;
		COMx.iBYTES_TO_SEND:=5;
		TXBuf[0]:=16#10;
		TXBuf[1]:=16#40;
		TXBuf[2]:=maddress;
		mchk:=TXBuf[1]+TXBuf[2];
		TXBuf[3]:=mchk;
		TXBuf[4]:=16#16;
		xSND:=TRUE;
	END_IF

	IF mt2 THEN
		mt2:=FALSE;
		COMx.iBYTES_TO_SEND:=9;
		TXBuf[0]:=16#68;
		TXBuf[1]:=16#03;
		TXBuf[2]:=16#03;
		TXBuf[3]:=16#68;
		TXBuf[4]:=16#53;
		TXBuf[5]:=maddress;
		TXBuf[6]:=16#BB;
		mchk:=TXBuf[4]+TXBuf[5]+TXBuf[6];
		TXBuf[7]:=mchk;
		TXBuf[8]:=16#16;
		xSND:=TRUE;
	END_IF

	IF mt3 THEN
		mt3:=FALSE;
		COMx.iBYTES_TO_SEND:=5;
		TXBuf[0]:=16#10;
		TXBuf[1]:=16#5B;
		TXBuf[2]:=maddress;
		mchk:=TXBuf[1]+TXBuf[2];
		TXBuf[3]:=mchk;
		TXBuf[4]:=16#16;
		xSND:=TRUE;
	END_IF
*)

END_IF


IF delFileIdx THEN
		SysFileDelete('S:\LOG.IDX');
END_IF
(*==============================*)
(*== System cycle operations ===*)
(*==============================*)
(* Execute TCP processes *)

Logger_Proc(); 
Remote_Proc();


(* Update user led *)
USRLED_Update();
(* Execute Cron Editor commands *)
CronEd();
(*...*)
(* External resources *)
IF TPV01.ERR THEN T_AMB:=Plant_DefaultTAmb; ELSE T_AMB:=TT_S01; END_IF

(**** SIMULATION ONLY ****)
(*...*)
END_PROGRAM
ACTION Main_Stm:
CASE Sys.Status OF
	(*--------------------------------------------------------*)
	S_STARTUP:
		Sys.Status:=S_INIT_RTC;
	(*--------------------------------------------------------*)
	S_INIT_RTC:
		(* Check RTC and update from network *)
		RTC_Update();
		(* Check time *)
		IF Sys.Time_Year>2000 THEN
			Sys.Status:=S_INIT_VAR;
		END_IF
	(*--------------------------------------------------------*)
	S_INIT_VAR:
		LogEv(EL_Wrn,EO_SYS,0,1,CONCAT('System_startup_v',WORD_TO_STRING(Plant_SW_VER)));
		Sys.Status:=S_RUNNING;
	(*--------------------------------------------------------*)
	S_RUNNING:

		Timer1(IN:=NOT Timer1.Q,PT:=T#150ms);
		IF Timer1.Q THEN
			(* Update system checks *)
			SCA_Proc();
			SYS_Proc();
		END_IF

		Timer2(IN:=NOT Timer2.Q,PT:=T#500ms);
		IF Timer2.Q THEN
			(* Read current date/time *)
			RTC_Update();
			(* === Execute plant operations === *)
			(* Temperature da RTD *)
			TPV01	 ( IN:=TT_S01 );
			(* Temperature da Convertitori 4-20mA *)
			TPV02	 ( AI_INPUT:=TT_S02 );
			TPV03	 ( AI_INPUT:=TT_S03 );
			TPV04	 ( AI_INPUT:=TT_S04 );
			TPV05	 ( AI_INPUT:=TT_S05 );
			TPV06	 ( AI_INPUT:=TT_S06 );
			TPV07	 ( AI_INPUT:=TT_S07 );
			TPV08	 ( AI_INPUT:=TT_S08 );
			TPV09	 ( AI_INPUT:=TT_S09 );



			(* Contabilizzatori Digitali *)
				(* Media dinamica delle temperature valide *)
				t_sum:=0; t_cnt:=0;
				IF NOT TPV02.ERR THEN t_sum:=t_sum+TPV02.ValoreScalato; t_cnt:=t_cnt+1; END_IF
				IF NOT TPV03.ERR THEN t_sum:=t_sum+TPV03.ValoreScalato; t_cnt:=t_cnt+1; END_IF
				IF NOT TPV04.ERR THEN t_sum:=t_sum+TPV04.ValoreScalato; t_cnt:=t_cnt+1; END_IF
				IF t_cnt>0 THEN CTB250.T_SEND:=t_sum/t_cnt; ELSE CTB250.T_SEND:=-9999; END_IF
				t_sum:=0; t_cnt:=0;
				IF NOT TPV05.ERR THEN t_sum:=t_sum+TPV05.ValoreScalato; t_cnt:=t_cnt+1; END_IF
				IF NOT TPV06.ERR THEN t_sum:=t_sum+TPV06.ValoreScalato; t_cnt:=t_cnt+1; END_IF
				IF NOT TPV07.ERR THEN t_sum:=t_sum+TPV07.ValoreScalato; t_cnt:=t_cnt+1; END_IF
				IF t_cnt>0 THEN CTB250.T_RET:=t_sum/t_cnt; ELSE CTB250.T_RET:=-9999; END_IF

				(* Ferma contabilizzazione se manca una temperatura *)
				IF CTB250.T_SEND=-9999 OR CTB250.T_RET=-9999 THEN CTB250.T_SEND:=0; CTB250.T_RET:=0; END_IF
			CTB250   (	FLOW  :=PORT01.ValoreScalato,
						ENERGY_WH:=CTB250_ENERGY_WH,
						ENERGY   :=CTB250_ENERGY );




			(* Crono  *)
			THER01();
			CIRD01.OnOff:=THER01.RunCrono; (* Circolatore P2 - P3 *)
			THER02();
			CIRD02.OnOff:=THER02.RunCrono; (* Circolatore P4 - P5 *)
			THER03();
			EV02.OnOff:=THER03.RunCrono; (* Comando EV02 che asserve lacaldia CAL02 *)
			THER04();
			EV03.OnOff:=THER04.RunCrono; (* Comando EV03 che asserve lacaldia CAL03 *)


			(* Caldaia in RUN *)

			DelayOffPompe(IN:=CIRD01.PumpA_ST
							OR CIRD01.PumpB_ST
							OR CIRD02.PumpA_ST
							OR CIRD02.PumpB_ST,PT:=t#10s);


			CAL02.Run := 	THER03.RunCrono  		(* comano da crono *)
							AND EV02.EV_Open		(* Elettrovalvola Aperta *)
							AND DelayOffPompe.Q
							AND SCA_Proc.SCA04_14.OUT (* Valvola Vaso Espansione aperto *)
							;

			(* Set Point Caldaia *)
			OffsetSetPointManuale:=0; (* in questo impianto non c'è scambiatore *)
			CAL02.SetPointManuale:=THER03.SetPoint - OffsetSetPointManuale;
			CAL02.AbilitaSetPointManuale:=TRUE;


			CAL03.Run := 	THER04.RunCrono  		(* comano da crono *)
							AND EV03.EV_Open		(* Elettrovalvola Aperta *)
							AND DelayOffPompe.Q
							AND SCA_Proc.SCA05_14.OUT (* Valvola Vaso Espansione aperto *)
							;

			(* Set Point Caldaia *)
			OffsetSetPointManuale:=0; (* in questo impianto non c'è scambiatore *)
			CAL03.SetPointManuale:=THER04.SetPoint - OffsetSetPointManuale;
			CAL03.AbilitaSetPointManuale:=TRUE;





			(* Test toggle *)
			IF TEST1 THEN TEST1:=FALSE; ELSE TEST1:=TRUE; END_IF
		     END_IF

		Timer3(IN:=NOT Timer3.Q,PT:=T#5m);
		IF Timer3.Q OR SendLog THEN
			(* Trig logger *)
			LogTrig();
			(* Execute temporary CSV logger *)
			CSV_Log();
		END_IF

		(* Contabilizzatori Digitali *)
		PORT01( DI_Input:=PORT01_DI, AI_INPUT:=PORT01_AI,
				Totalizzatore:=PortataTotalePORT01,
				Contatore:=ConteggioTotalePORT01 );


	(*--------------------------------------------------------*)
	S_SHUTDOWN:
		(* Arresto del sistema *)
		Sys.Status:=S_STARTUP;
	(*--------------------------------------------------------*)
	S_HALT:
		(* Aspetta uscita manuale *)
		Sys.Status:=S_STARTUP;
	(*--------------------------------------------------------*)
ELSE
	Sys.Status:=S_STARTUP;
END_CASE;
END_ACTION

(* POU Plant/SCA_Proc, ST *)
PROGRAM SCA_Proc
VAR
	SCA01_5			:FLT_TAP;
	SCA01_6			:FLT_TAP;

(*	SCA02_1			:FLT_TAP;
	SCA02_2			:FLT_TAP;
	SCA02_3			:FLT_TAP;
	SCA02_4			:FLT_TAP;
	SCA02_5			:FLT_TAP;
	SCA02_6			:FLT_TAP;
	SCA02_7			:FLT_TAP;
	SCA02_8			:FLT_TAP;
	SCA02_9			:FLT_TAP;

	SCA03_1			:FLT_TAP;
	SCA03_2			:FLT_TAP;
	SCA03_3			:FLT_TAP;
	SCA03_4			:FLT_TAP;
	SCA03_5			:FLT_TAP;
	SCA03_6			:FLT_TAP;
	SCA03_7			:FLT_TAP;
	SCA03_8			:FLT_TAP;
	SCA03_9			:FLT_TAP;
	SCA03_10		:FLT_TAP;
	SCA03_11		:FLT_TAP;
	SCA03_12		:FLT_TAP;
	SCA03_13		:FLT_TAP;
	SCA03_14		:FLT_TAP;
	SCA03_15		:FLT_TAP;
	SCA03_16		:FLT_TAP;
	SCA03_17		:FLT_TAP;
	SCA03_18		:FLT_TAP;
	SCA03_19		:FLT_TAP;
	SCA03_20		:FLT_TAP;
	SCA03_21		:FLT_TAP;
	SCA03_22		:FLT_TAP;
*)


	SCA04_1			:FLT_TAP;
	SCA04_2			:FLT_TAP;
	SCA04_3			:FLT_TAP;
	SCA04_4			:FLT_TAP;
	SCA04_5			:FLT_TAP;
	SCA04_6			:FLT_TAP;
	SCA04_7			:FLT_TAP;
	SCA04_8			:FLT_TAP;
	SCA04_9			:FLT_TAP;
	SCA04_10		:FLT_TAP;
	SCA04_11		:FLT_TAP;
	SCA04_12		:FLT_TAP;
	SCA04_13		:FLT_TAP;
	SCA04_14		:FLT_TAP;

	SCA05_1			:FLT_TAP;
	SCA05_2			:FLT_TAP;
	SCA05_3			:FLT_TAP;
	SCA05_4			:FLT_TAP;
	SCA05_5			:FLT_TAP;
	SCA05_6			:FLT_TAP;
	SCA05_7			:FLT_TAP;
	SCA05_8			:FLT_TAP;
	SCA05_9			:FLT_TAP;
	SCA05_10		:FLT_TAP;
	SCA05_11		:FLT_TAP;
	SCA05_12		:FLT_TAP;
	SCA05_13		:FLT_TAP;
	SCA05_14		:FLT_TAP;

	SCA06_1			:FLT_TAP;
	SCA06_2			:FLT_TAP;
	SCA06_3			:FLT_TAP;
	SCA06_4			:FLT_TAP;
	SCA06_5			:FLT_TAP;
	SCA06_6			:FLT_TAP;
	SCA06_7			:FLT_TAP;
	SCA06_8			:FLT_TAP;
	SCA06_9			:FLT_TAP;
	SCA06_10		:FLT_TAP;
	SCA06_11		:FLT_TAP;
	SCA06_12		:FLT_TAP;


	SCA06_15		:FLT_TAP;
	SCA06_16		:FLT_TAP;
	SCA06_17		:FLT_TAP;
	SCA06_18		:FLT_TAP;
	SCA06_19		:FLT_TAP;
	SCA06_20		:FLT_TAP;
	SCA06_21		:FLT_TAP;
	SCA06_22		:FLT_TAP;







	upd : BOOL;
END_VAR
(***** SCA01 *****)
SCA01_1_DO:=SCA01_6.OUT; (* Comando - messaggio vocale su SCA01.6 *)

SCA01_2_DO:=SCA05_1.OUT OR SCA04_1.OUT;

SCA01_3_DO:=	SCA04_3.OUT  OR SCA04_4.OUT  OR SCA04_5.OUT  OR
			 	SCA04_6.OUT  OR SCA04_7.OUT  OR SCA04_8.OUT  OR
				SCA04_9.OUT  OR SCA04_10.OUT OR SCA04_11.OUT OR
				SCA05_3.OUT  OR SCA05_4.OUT  OR SCA05_5.OUT OR
				SCA05_6.OUT  OR SCA05_7.OUT  OR SCA05_8.OUT OR
				SCA05_9.OUT  OR SCA05_10.OUT OR SCA05_11.OUT
				;

SCA01_4_DO:=SCA06_1.OUT  OR SCA06_2.OUT  OR SCA06_6.OUT  OR
			SCA06_8.OUT OR SCA06_10.OUT OR
			SCA06_16.OUT OR SCA06_12.OUT OR SCA06_20.OUT OR
			NOT CIRD01A_AL OR NOT CIRD01B_AL OR NOT CIRD02A_AL OR NOT CIRD02B_AL
			;
(*
SCA01_3_DO:=SCA02_3.OUT  OR SCA02_4.OUT  OR SCA02_5.OUT  OR SCA02_6.OUT  OR
			SCA02_8.OUT  OR SCA02_9.OUT;

SCA01_4_DO:=SCA03_1.OUT  OR SCA03_2.OUT  OR SCA03_4.OUT  OR SCA03_6.OUT  OR
			SCA03_8.OUT  OR SCA03_10.OUT OR SCA03_12.OUT OR SCA03_14.OUT OR
			SCA03_16.OUT OR SCA03_18.OUT OR SCA03_20.OUT OR SCA03_22.OUT;
*)







SCA01_5(IN:=NOT SCA01_5_DI);
IF SCA01_5.EVL THEN LogEv(EL_Log,EO_SCA,1,0,'5'); upd:=TRUE; END_IF
IF SCA01_5.EVH THEN	LogEv(EL_Log,EO_SCA,1,1,'5'); upd:=TRUE; END_IF

SCA01_6(IN:=NOT SCA01_6_DI);
IF SCA01_6.EVL THEN	LogEv(EL_Log,EO_SCA,1,0,'6'); upd:=TRUE; END_IF
IF SCA01_6.EVH THEN	LogEv(EL_Log,EO_SCA,1,1,'6'); upd:=TRUE; END_IF

(***** SCA04 *****)

SCA04_1(IN:= NOT SCA04_1_DI);  (* Caldaia IN fUNZIONE *)
IF SCA04_1.EVL THEN	LogEv(EL_Log,EO_SCA,4,0,'1'); upd:=TRUE; END_IF
IF SCA04_1.EVH THEN	LogEv(EL_Log,EO_SCA,4,1,'1'); upd:=TRUE; END_IF
SCA04_2(IN:=SCA04_2_DI);
IF SCA04_2.EVL THEN	LogEv(EL_Log,EO_SCA,4,0,'2'); Upd:=TRUE; END_IF
IF SCA04_2.EVH THEN	LogEv(EL_Log,EO_SCA,4,1,'2'); upd:=TRUE; END_IF
SCA04_3(IN:=NOT SCA04_3_DI);
IF SCA04_3.EVH THEN	LogEv(EL_Log,EO_SCA,4,1,'3'); upd:=TRUE; END_IF
IF SCA04_3.EVL THEN	LogEv(EL_Log,EO_SCA,4,0,'3'); upd:=TRUE; END_IF
SCA04_4(IN:=NOT SCA04_4_DI);
IF SCA04_4.EVH THEN	LogEv(EL_Log,EO_SCA,4,1,'4'); upd:=TRUE; END_IF
IF SCA04_4.EVL THEN	LogEv(EL_Log,EO_SCA,4,0,'4'); upd:=TRUE; END_IF
SCA04_5(IN:= SCA04_5_DI);
IF SCA04_5.EVH THEN	LogEv(EL_Log,EO_SCA,4,1,'5'); upd:=TRUE; END_IF
IF SCA04_5.EVL THEN	LogEv(EL_Log,EO_SCA,4,0,'5'); upd:=TRUE; END_IF
SCA04_6(IN:= SCA04_6_DI);
IF SCA04_6.EVH THEN	LogEv(EL_Log,EO_SCA,4,1,'6'); upd:=TRUE; END_IF
IF SCA04_6.EVL THEN	LogEv(EL_Log,EO_SCA,4,0,'6'); upd:=TRUE; END_IF
SCA04_7(IN:= SCA04_7_DI);
IF SCA04_7.EVH THEN	LogEv(EL_Log,EO_SCA,4,1,'7'); upd:=TRUE; END_IF
IF SCA04_7.EVL THEN	LogEv(EL_Log,EO_SCA,4,0,'7'); upd:=TRUE; END_IF
SCA04_8(IN:= SCA04_8_DI);
IF SCA04_8.EVH THEN	LogEv(EL_Log,EO_SCA,4,1,'8'); upd:=TRUE; END_IF
IF SCA04_8.EVL THEN	LogEv(EL_Log,EO_SCA,4,0,'8'); upd:=TRUE; END_IF
SCA04_9(IN:= SCA04_9_DI);
IF SCA04_9.EVH THEN	LogEv(EL_Log,EO_SCA,4,1,'9'); upd:=TRUE; END_IF
IF SCA04_9.EVL THEN	LogEv(EL_Log,EO_SCA,4,0,'9'); upd:=TRUE; END_IF
SCA04_10(IN:= SCA04_10_DI);
IF SCA04_10.EVH THEN LogEv(EL_Log,EO_SCA,4,1,'10'); upd:=TRUE; END_IF
IF SCA04_10.EVL THEN LogEv(EL_Log,EO_SCA,4,0,'10'); upd:=TRUE; END_IF
SCA04_11(IN:= NOT SCA04_11_DI);
IF SCA04_11.EVH THEN LogEv(EL_Log,EO_SCA,4,1,'11'); upd:=TRUE; END_IF
IF SCA04_11.EVL THEN LogEv(EL_Log,EO_SCA,4,0,'11'); upd:=TRUE; END_IF
SCA04_12(IN:= SCA04_12_DI);
IF SCA04_12.EVH THEN LogEv(EL_Log,EO_SCA,4,1,'12'); upd:=TRUE; END_IF
IF SCA04_12.EVL THEN LogEv(EL_Log,EO_SCA,4,0,'12'); upd:=TRUE; END_IF
SCA04_13(IN:= SCA04_13_DI);
IF SCA04_13.EVH THEN LogEv(EL_Log,EO_SCA,4,1,'13'); upd:=TRUE; END_IF
IF SCA04_13.EVL THEN LogEv(EL_Log,EO_SCA,4,0,'13'); upd:=TRUE; END_IF
SCA04_14(IN:= SCA04_14_DI);
IF SCA04_14.EVL THEN LogEv(EL_Log,EO_SCA,4,0,'14'); upd:=TRUE; END_IF
IF SCA04_14.EVH THEN LogEv(EL_Log,EO_SCA,4,1,'14'); upd:=TRUE; END_IF

(***** SCA05 *****)

SCA05_1(IN:= NOT SCA05_1_DI);   (* Caldaia IN fUNZIONE *)
IF SCA05_1.EVL THEN	LogEv(EL_Log,EO_SCA,5,0,'1'); upd:=TRUE; END_IF
IF SCA05_1.EVH THEN	LogEv(EL_Log,EO_SCA,5,1,'1'); upd:=TRUE; END_IF
SCA05_2(IN:=SCA05_2_DI);
IF SCA05_2.EVL THEN	LogEv(EL_Log,EO_SCA,5,0,'2'); Upd:=TRUE; END_IF
IF SCA05_2.EVH THEN	LogEv(EL_Log,EO_SCA,5,1,'2'); upd:=TRUE; END_IF
SCA05_3(IN:=NOT SCA05_3_DI);
IF SCA05_3.EVH THEN	LogEv(EL_Log,EO_SCA,5,1,'3'); upd:=TRUE; END_IF
IF SCA05_3.EVL THEN	LogEv(EL_Log,EO_SCA,5,0,'3'); upd:=TRUE; END_IF
SCA05_4(IN:=NOT SCA05_4_DI);
IF SCA05_4.EVH THEN	LogEv(EL_Log,EO_SCA,5,1,'4'); upd:=TRUE; END_IF
IF SCA05_4.EVL THEN	LogEv(EL_Log,EO_SCA,5,0,'4'); upd:=TRUE; END_IF
SCA05_5(IN:= SCA05_5_DI);
IF SCA05_5.EVH THEN	LogEv(EL_Log,EO_SCA,5,1,'5'); upd:=TRUE; END_IF
IF SCA05_5.EVL THEN	LogEv(EL_Log,EO_SCA,5,0,'5'); upd:=TRUE; END_IF
SCA05_6(IN:= SCA05_6_DI);
IF SCA05_6.EVH THEN	LogEv(EL_Log,EO_SCA,5,1,'6'); upd:=TRUE; END_IF
IF SCA05_6.EVL THEN	LogEv(EL_Log,EO_SCA,5,0,'6'); upd:=TRUE; END_IF
SCA05_7(IN:=  SCA05_7_DI);
IF SCA05_7.EVH THEN	LogEv(EL_Log,EO_SCA,5,1,'7'); upd:=TRUE; END_IF
IF SCA05_7.EVL THEN	LogEv(EL_Log,EO_SCA,5,0,'7'); upd:=TRUE; END_IF
SCA05_8(IN:= SCA05_8_DI);
IF SCA05_8.EVH THEN	LogEv(EL_Log,EO_SCA,5,1,'8'); upd:=TRUE; END_IF
IF SCA05_8.EVL THEN	LogEv(EL_Log,EO_SCA,5,0,'8'); upd:=TRUE; END_IF
SCA05_9(IN:= SCA05_9_DI);
IF SCA05_9.EVH THEN	LogEv(EL_Log,EO_SCA,5,1,'9'); upd:=TRUE; END_IF
IF SCA05_9.EVL THEN	LogEv(EL_Log,EO_SCA,5,0,'9'); upd:=TRUE; END_IF
SCA05_10(IN:= SCA05_10_DI);
IF SCA05_10.EVH THEN LogEv(EL_Log,EO_SCA,5,1,'10'); upd:=TRUE; END_IF
IF SCA05_10.EVL THEN LogEv(EL_Log,EO_SCA,5,0,'10'); upd:=TRUE; END_IF
SCA05_11(IN:= NOT SCA05_11_DI);
IF SCA05_11.EVH THEN LogEv(EL_Log,EO_SCA,5,1,'11'); upd:=TRUE; END_IF
IF SCA05_11.EVL THEN LogEv(EL_Log,EO_SCA,5,0,'11'); upd:=TRUE; END_IF
SCA05_12(IN:= SCA05_12_DI);
IF SCA05_12.EVL THEN LogEv(EL_Log,EO_SCA,5,0,'12'); upd:=TRUE; END_IF
IF SCA05_12.EVH THEN LogEv(EL_Log,EO_SCA,5,1,'12'); upd:=TRUE; END_IF
SCA05_13(IN:= SCA05_13_DI);
IF SCA05_13.EVL THEN LogEv(EL_Log,EO_SCA,5,0,'13'); upd:=TRUE; END_IF
IF SCA05_13.EVH THEN LogEv(EL_Log,EO_SCA,5,1,'13'); upd:=TRUE; END_IF
SCA05_14(IN:=SCA05_14_DI);
IF SCA05_14.EVH THEN LogEv(EL_Log,EO_SCA,5,1,'14'); upd:=TRUE; END_IF
IF SCA05_14.EVL THEN LogEv(EL_Log,EO_SCA,5,0,'14'); upd:=TRUE; END_IF


(***** SCA06 *****)

SCA06_1(IN:=NOT SCA06_1_DI);
IF SCA06_1.EVL THEN	LogEv(EL_Wrn,EO_SCA,6,0,'1'); upd:=TRUE; END_IF
IF SCA06_1.EVH THEN	LogEv(EL_Log,EO_SCA,6,1,'1'); upd:=TRUE; END_IF
SCA06_2(IN:=NOT SCA06_2_DI);
IF SCA06_2.EVL THEN	LogEv(EL_Log,EO_SCA,6,0,'2'); Upd:=TRUE; END_IF
IF SCA06_2.EVH THEN	LogEv(EL_Log,EO_SCA,6,1,'2'); upd:=TRUE; END_IF
SCA06_3(IN:= SCA06_3_DI);
IF SCA06_3.EVL THEN	LogEv(EL_Wrn,EO_SCA,6,0,'3'); upd:=TRUE; END_IF
IF SCA06_3.EVH THEN	LogEv(EL_Log,EO_SCA,6,1,'3'); upd:=TRUE; END_IF
SCA06_4(IN:= SCA06_4_DI);
IF SCA06_4.EVL THEN	LogEv(EL_Wrn,EO_SCA,6,0,'4'); upd:=TRUE; END_IF
IF SCA06_4.EVH THEN	LogEv(EL_Log,EO_SCA,6,1,'4'); upd:=TRUE; END_IF
SCA06_5(IN:= SCA06_5_DI);
IF SCA06_5.EVL THEN	LogEv(EL_Log,EO_SCA,6,0,'5'); upd:=TRUE; END_IF
IF SCA06_5.EVH THEN	LogEv(EL_Log,EO_SCA,6,1,'5'); upd:=TRUE; END_IF
SCA06_6(IN:=NOT SCA06_6_DI);
IF SCA06_6.EVL THEN	LogEv(EL_Wrn,EO_SCA,6,0,'6'); upd:=TRUE; END_IF
IF SCA06_6.EVH THEN	LogEv(EL_Log,EO_SCA,6,1,'6'); upd:=TRUE; END_IF
SCA06_7(IN:=SCA06_7_DI);
IF SCA06_7.EVL THEN	LogEv(EL_Log,EO_SCA,6,0,'7'); upd:=TRUE; END_IF
IF SCA06_7.EVH THEN	LogEv(EL_Log,EO_SCA,6,1,'7'); upd:=TRUE; END_IF
SCA06_8(IN:=NOT SCA06_8_DI);
IF SCA06_8.EVL THEN	LogEv(EL_Wrn,EO_SCA,6,0,'8'); upd:=TRUE; END_IF
IF SCA06_8.EVH THEN	LogEv(EL_Log,EO_SCA,6,1,'8'); upd:=TRUE; END_IF
SCA06_9(IN:= SCA06_9_DI);
IF SCA06_9.EVL THEN	LogEv(EL_Log,EO_SCA,6,0,'9'); upd:=TRUE; END_IF
IF SCA06_9.EVH THEN	LogEv(EL_Log,EO_SCA,6,1,'9'); upd:=TRUE; END_IF
SCA06_10(IN:=NOT SCA06_10_DI);
IF SCA06_10.EVL THEN LogEv(EL_Wrn,EO_SCA,6,0,'10'); upd:=TRUE; END_IF
IF SCA06_10.EVH THEN LogEv(EL_Log,EO_SCA,6,1,'10'); upd:=TRUE; END_IF
SCA06_11(IN:= SCA06_11_DI);
IF SCA06_11.EVL THEN	LogEv(EL_Log,EO_SCA,6,0,'11'); upd:=TRUE; END_IF
IF SCA06_11.EVH THEN	LogEv(EL_Log,EO_SCA,6,1,'11'); upd:=TRUE; END_IF
SCA06_12(IN:=NOT SCA06_12_DI);
IF SCA06_12.EVL THEN	LogEv(EL_Wrn,EO_SCA,6,0,'12'); Upd:=TRUE; END_IF
IF SCA06_12.EVH THEN	LogEv(EL_Log,EO_SCA,6,1,'12'); upd:=TRUE; END_IF



SCA06_15(IN:= SCA06_15_DI);
IF SCA06_15.EVL THEN	LogEv(EL_Log,EO_SCA,6,0,'15'); upd:=TRUE; END_IF
IF SCA06_15.EVH THEN	LogEv(EL_Log,EO_SCA,6,1,'15'); upd:=TRUE; END_IF
SCA06_16(IN:=NOT SCA06_16_DI);
IF SCA06_16.EVL THEN	LogEv(EL_Wrn,EO_SCA,6,0,'16'); upd:=TRUE; END_IF
IF SCA06_16.EVH THEN	LogEv(EL_Log,EO_SCA,6,1,'16'); upd:=TRUE; END_IF
(*
SCA06_17(IN:=SCA06_17_DI);
IF SCA06_17.EVL THEN	LogEv(EL_Log,EO_SCA,6,1,'17'); upd:=TRUE; END_IF
IF SCA06_17.EVH THEN	LogEv(EL_Log,EO_SCA,6,2,'17'); upd:=TRUE; END_IF
SCA06_18(IN:= SCA06_18_DI);
IF SCA06_18.EVL THEN	LogEv(EL_Wrn,EO_SCA,6,1,'18'); upd:=TRUE; END_IF
IF SCA06_18.EVH THEN	LogEv(EL_Log,EO_SCA,6,2,'18'); upd:=TRUE; END_IF
*)
SCA06_19(IN:= SCA06_19_DI);
IF SCA06_19.EVL THEN	LogEv(EL_Log,EO_SCA,6,0,'19'); upd:=TRUE; END_IF
IF SCA06_19.EVH THEN	LogEv(EL_Log,EO_SCA,6,1,'19'); upd:=TRUE; END_IF
SCA06_20(IN:=NOT SCA06_20_DI);
IF SCA06_20.EVL THEN LogEv(EL_Wrn,EO_SCA,6,0,'20'); upd:=TRUE; END_IF
IF SCA06_20.EVH THEN LogEv(EL_Log,EO_SCA,6,1,'20'); upd:=TRUE; END_IF
SCA06_21(IN:= SCA06_21_DI);
IF SCA06_21.EVL THEN	LogEv(EL_Wrn,EO_SCA,6,0,'21'); upd:=TRUE; END_IF
IF SCA06_21.EVH THEN	LogEv(EL_Log,EO_SCA,6,1,'21'); upd:=TRUE; END_IF
SCA06_22(IN:=SCA06_22_DI);
IF SCA06_22.EVL THEN	LogEv(EL_Log,EO_SCA,6,0,'22'); Upd:=TRUE; END_IF
IF SCA06_22.EVH THEN	LogEv(EL_Log,EO_SCA,6,1,'22'); upd:=TRUE; END_IF


(*

(***** SCA03 *****)

SCA03_1(IN:=NOT SCA03_1_DI);
IF SCA03_1.EVL THEN	LogEv(EL_Wrn,EO_SCA,3,1,'1'); upd:=TRUE; END_IF
IF SCA03_1.EVH THEN	LogEv(EL_Log,EO_SCA,3,2,'1'); upd:=TRUE; END_IF
SCA03_2(IN:=NOT SCA03_2_DI);
IF SCA03_2.EVL THEN	LogEv(EL_Wrn,EO_SCA,3,1,'2'); upd:=TRUE; END_IF
IF SCA03_2.EVH THEN	LogEv(EL_Log,EO_SCA,3,2,'2'); upd:=TRUE; END_IF
SCA03_3(IN:=SCA03_3_DI);
IF SCA03_3.EVL THEN	LogEv(EL_Log,EO_SCA,3,1,'3'); END_IF
IF SCA03_3.EVH THEN	LogEv(EL_Log,EO_SCA,3,2,'3'); END_IF
SCA03_4(IN:=NOT SCA03_4_DI);
IF SCA03_4.EVL THEN	LogEv(EL_Wrn,EO_SCA,3,1,'4'); upd:=TRUE; END_IF
IF SCA03_4.EVH THEN	LogEv(EL_Log,EO_SCA,3,2,'4'); upd:=TRUE; END_IF
SCA03_5(IN:=SCA03_5_DI);
IF SCA03_5.EVL THEN	LogEv(EL_Log,EO_SCA,3,1,'5'); END_IF
IF SCA03_5.EVH THEN	LogEv(EL_Log,EO_SCA,3,2,'5'); END_IF
SCA03_6(IN:=NOT SCA03_6_DI);
IF SCA03_6.EVL THEN	LogEv(EL_Wrn,EO_SCA,3,1,'6'); upd:=TRUE; END_IF
IF SCA03_6.EVH THEN	LogEv(EL_Log,EO_SCA,3,2,'6'); upd:=TRUE; END_IF
SCA03_7(IN:=SCA03_7_DI);
IF SCA03_7.EVL THEN	LogEv(EL_Log,EO_SCA,3,1,'7'); END_IF
IF SCA03_7.EVH THEN	LogEv(EL_Log,EO_SCA,3,2,'7'); END_IF
SCA03_8(IN:=NOT SCA03_8_DI);
IF SCA03_8.EVL THEN	LogEv(EL_Wrn,EO_SCA,3,1,'8'); upd:=TRUE; END_IF
IF SCA03_8.EVH THEN	LogEv(EL_Log,EO_SCA,3,2,'8'); upd:=TRUE; END_IF
SCA03_9(IN:=SCA03_9_DI);
IF SCA03_9.EVL THEN	LogEv(EL_Log,EO_SCA,3,1,'9'); END_IF
IF SCA03_9.EVH THEN	LogEv(EL_Log,EO_SCA,3,2,'9'); END_IF
SCA03_10(IN:=NOT SCA03_10_DI);
IF SCA03_10.EVL THEN	LogEv(EL_Wrn,EO_SCA,3,1,'10'); upd:=TRUE; END_IF
IF SCA03_10.EVH THEN	LogEv(EL_Log,EO_SCA,3,2,'10'); upd:=TRUE; END_IF
SCA03_11(IN:=SCA03_11_DI);
IF SCA03_11.EVL THEN	LogEv(EL_Log,EO_SCA,3,1,'11'); END_IF
IF SCA03_11.EVH THEN	LogEv(EL_Log,EO_SCA,3,2,'11'); END_IF
SCA03_12(IN:=NOT SCA03_12_DI);
IF SCA03_12.EVL THEN	LogEv(EL_Wrn,EO_SCA,3,1,'12'); upd:=TRUE; END_IF
IF SCA03_12.EVH THEN	LogEv(EL_Log,EO_SCA,3,2,'12'); upd:=TRUE; END_IF
SCA03_13(IN:=SCA03_13_DI);
IF SCA03_13.EVL THEN	LogEv(EL_Log,EO_SCA,3,1,'13'); END_IF
IF SCA03_13.EVH THEN	LogEv(EL_Log,EO_SCA,3,2,'13'); END_IF
SCA03_14(IN:=NOT SCA03_14_DI);
IF SCA03_14.EVL THEN	LogEv(EL_Wrn,EO_SCA,3,1,'14'); upd:=TRUE; END_IF
IF SCA03_14.EVH THEN	LogEv(EL_Log,EO_SCA,3,2,'14'); upd:=TRUE; END_IF
SCA03_15(IN:=SCA03_15_DI);
IF SCA03_15.EVL THEN	LogEv(EL_Log,EO_SCA,3,1,'15'); END_IF
IF SCA03_15.EVH THEN	LogEv(EL_Log,EO_SCA,3,2,'15'); END_IF
SCA03_16(IN:=NOT SCA03_16_DI);
IF SCA03_16.EVL THEN	LogEv(EL_Wrn,EO_SCA,3,1,'16'); upd:=TRUE; END_IF
IF SCA03_16.EVH THEN	LogEv(EL_Log,EO_SCA,3,2,'16'); upd:=TRUE; END_IF
SCA03_17(IN:=SCA03_17_DI);
IF SCA03_17.EVL THEN	LogEv(EL_Log,EO_SCA,3,1,'17'); END_IF
IF SCA03_17.EVH THEN	LogEv(EL_Log,EO_SCA,3,2,'17'); END_IF
SCA03_18(IN:=NOT SCA03_18_DI);
IF SCA03_18.EVL THEN	LogEv(EL_Wrn,EO_SCA,3,1,'18'); upd:=TRUE; END_IF
IF SCA03_18.EVH THEN	LogEv(EL_Log,EO_SCA,3,2,'18'); upd:=TRUE; END_IF
SCA03_19(IN:=SCA03_19_DI);
IF SCA03_19.EVL THEN	LogEv(EL_Log,EO_SCA,3,1,'19'); END_IF
IF SCA03_19.EVH THEN	LogEv(EL_Log,EO_SCA,3,2,'19'); END_IF
SCA03_20(IN:=NOT SCA03_20_DI);
IF SCA03_20.EVL THEN	LogEv(EL_Wrn,EO_SCA,3,1,'20'); upd:=TRUE; END_IF
IF SCA03_20.EVH THEN	LogEv(EL_Log,EO_SCA,3,2,'20'); upd:=TRUE; END_IF
SCA03_21(IN:=SCA03_21_DI);
IF SCA03_21.EVL THEN	LogEv(EL_Log,EO_SCA,3,1,'21'); END_IF
IF SCA03_21.EVH THEN	LogEv(EL_Log,EO_SCA,3,2,'21'); END_IF
SCA03_22(IN:=NOT SCA03_22_DI);
IF SCA03_22.EVL THEN	LogEv(EL_Wrn,EO_SCA,3,1,'22'); upd:=TRUE; END_IF
IF SCA03_22.EVH THEN	LogEv(EL_Log,EO_SCA,3,2,'22'); upd:=TRUE; END_IF

*)



IF upd THEN
	upd:=FALSE;
	Logger_Head();
	AddLogData();
	Logger_Send();
END_IF
END_PROGRAM
ACTION AddLogData:
Logger.s1:='&SCA01=';
Logger.s1:=CONCAT(Logger.s1,BYTE_TO_STRING(BOOL_TO_BYTE(SCA01_1_DO))		); Logger.s1:=CONCAT(Logger.s1,';');
Logger.s1:=CONCAT(Logger.s1,BYTE_TO_STRING(BOOL_TO_BYTE(SCA01_2_DO))		); Logger.s1:=CONCAT(Logger.s1,';');
Logger.s1:=CONCAT(Logger.s1,BYTE_TO_STRING(BOOL_TO_BYTE(SCA01_3_DO))		); Logger.s1:=CONCAT(Logger.s1,';');
Logger.s1:=CONCAT(Logger.s1,BYTE_TO_STRING(BOOL_TO_BYTE(SCA01_4_DO))		); Logger.s1:=CONCAT(Logger.s1,';');
Logger.s1:=CONCAT(Logger.s1,BYTE_TO_STRING(BOOL_TO_BYTE(SCA01_5.OUT))		); Logger.s1:=CONCAT(Logger.s1,';');
Logger.s1:=CONCAT(Logger.s1,BYTE_TO_STRING(BOOL_TO_BYTE(SCA01_6.OUT))		);
ADDSTRING(ADR(Logger.TData), ADR(Logger.s1), Logger.TLen);

Logger.s1:='&SCA04=';
Logger.s1:=CONCAT(Logger.s1,BYTE_TO_STRING(BOOL_TO_BYTE(SCA04_1.OUT))		); Logger.s1:=CONCAT(Logger.s1,';');
Logger.s1:=CONCAT(Logger.s1,BYTE_TO_STRING(BOOL_TO_BYTE(SCA04_2.OUT))		); Logger.s1:=CONCAT(Logger.s1,';');
Logger.s1:=CONCAT(Logger.s1,BYTE_TO_STRING(BOOL_TO_BYTE(SCA04_3.OUT))		); Logger.s1:=CONCAT(Logger.s1,';');
Logger.s1:=CONCAT(Logger.s1,BYTE_TO_STRING(BOOL_TO_BYTE(SCA04_4.OUT))		); Logger.s1:=CONCAT(Logger.s1,';');
Logger.s1:=CONCAT(Logger.s1,BYTE_TO_STRING(BOOL_TO_BYTE(SCA04_5.OUT))		); Logger.s1:=CONCAT(Logger.s1,';');
Logger.s1:=CONCAT(Logger.s1,BYTE_TO_STRING(BOOL_TO_BYTE(SCA04_6.OUT))		); Logger.s1:=CONCAT(Logger.s1,';');
Logger.s1:=CONCAT(Logger.s1,BYTE_TO_STRING(BOOL_TO_BYTE(SCA04_7.OUT))		); Logger.s1:=CONCAT(Logger.s1,';');
Logger.s1:=CONCAT(Logger.s1,BYTE_TO_STRING(BOOL_TO_BYTE(SCA04_8.OUT))		); Logger.s1:=CONCAT(Logger.s1,';');
Logger.s1:=CONCAT(Logger.s1,BYTE_TO_STRING(BOOL_TO_BYTE(SCA04_9.OUT))		); Logger.s1:=CONCAT(Logger.s1,';');
Logger.s1:=CONCAT(Logger.s1,BYTE_TO_STRING(BOOL_TO_BYTE(SCA04_10.OUT))		); Logger.s1:=CONCAT(Logger.s1,';');
Logger.s1:=CONCAT(Logger.s1,BYTE_TO_STRING(BOOL_TO_BYTE(SCA04_11.OUT))		); Logger.s1:=CONCAT(Logger.s1,';');
Logger.s1:=CONCAT(Logger.s1,BYTE_TO_STRING(BOOL_TO_BYTE(SCA04_12.OUT))		); Logger.s1:=CONCAT(Logger.s1,';');
Logger.s1:=CONCAT(Logger.s1,BYTE_TO_STRING(BOOL_TO_BYTE(SCA04_13.OUT))		); Logger.s1:=CONCAT(Logger.s1,';');
Logger.s1:=CONCAT(Logger.s1,BYTE_TO_STRING(BOOL_TO_BYTE(SCA04_14.OUT))		);
ADDSTRING(ADR(Logger.TData), ADR(Logger.s1), Logger.TLen);

Logger.s1:='&SCA05=';
Logger.s1:=CONCAT(Logger.s1,BYTE_TO_STRING(BOOL_TO_BYTE(SCA05_1.OUT))		); Logger.s1:=CONCAT(Logger.s1,';');
Logger.s1:=CONCAT(Logger.s1,BYTE_TO_STRING(BOOL_TO_BYTE(SCA05_2.OUT))		); Logger.s1:=CONCAT(Logger.s1,';');
Logger.s1:=CONCAT(Logger.s1,BYTE_TO_STRING(BOOL_TO_BYTE(SCA05_3.OUT))		); Logger.s1:=CONCAT(Logger.s1,';');
Logger.s1:=CONCAT(Logger.s1,BYTE_TO_STRING(BOOL_TO_BYTE(SCA05_4.OUT))		); Logger.s1:=CONCAT(Logger.s1,';');
Logger.s1:=CONCAT(Logger.s1,BYTE_TO_STRING(BOOL_TO_BYTE(SCA05_5.OUT))		); Logger.s1:=CONCAT(Logger.s1,';');
Logger.s1:=CONCAT(Logger.s1,BYTE_TO_STRING(BOOL_TO_BYTE(SCA05_6.OUT))		); Logger.s1:=CONCAT(Logger.s1,';');
Logger.s1:=CONCAT(Logger.s1,BYTE_TO_STRING(BOOL_TO_BYTE(SCA05_7.OUT))		); Logger.s1:=CONCAT(Logger.s1,';');
Logger.s1:=CONCAT(Logger.s1,BYTE_TO_STRING(BOOL_TO_BYTE(SCA05_8.OUT))		); Logger.s1:=CONCAT(Logger.s1,';');
Logger.s1:=CONCAT(Logger.s1,BYTE_TO_STRING(BOOL_TO_BYTE(SCA05_9.OUT))		); Logger.s1:=CONCAT(Logger.s1,';');
Logger.s1:=CONCAT(Logger.s1,BYTE_TO_STRING(BOOL_TO_BYTE(SCA05_10.OUT))		); Logger.s1:=CONCAT(Logger.s1,';');
Logger.s1:=CONCAT(Logger.s1,BYTE_TO_STRING(BOOL_TO_BYTE(SCA05_11.OUT))		); Logger.s1:=CONCAT(Logger.s1,';');
Logger.s1:=CONCAT(Logger.s1,BYTE_TO_STRING(BOOL_TO_BYTE(SCA05_12.OUT))		); Logger.s1:=CONCAT(Logger.s1,';');
Logger.s1:=CONCAT(Logger.s1,BYTE_TO_STRING(BOOL_TO_BYTE(SCA05_13.OUT))		); Logger.s1:=CONCAT(Logger.s1,';');
Logger.s1:=CONCAT(Logger.s1,BYTE_TO_STRING(BOOL_TO_BYTE(SCA05_14.OUT))		);
ADDSTRING(ADR(Logger.TData), ADR(Logger.s1), Logger.TLen);

Logger.s1:='&SCA06=';
Logger.s1:=CONCAT(Logger.s1,BYTE_TO_STRING(BOOL_TO_BYTE(SCA06_1.OUT))		); Logger.s1:=CONCAT(Logger.s1,';');
Logger.s1:=CONCAT(Logger.s1,BYTE_TO_STRING(BOOL_TO_BYTE(SCA06_2.OUT))		); Logger.s1:=CONCAT(Logger.s1,';');
Logger.s1:=CONCAT(Logger.s1,BYTE_TO_STRING(BOOL_TO_BYTE(SCA06_3.OUT))		); Logger.s1:=CONCAT(Logger.s1,';');
Logger.s1:=CONCAT(Logger.s1,BYTE_TO_STRING(BOOL_TO_BYTE(SCA06_4.OUT))		); Logger.s1:=CONCAT(Logger.s1,';');
Logger.s1:=CONCAT(Logger.s1,BYTE_TO_STRING(BOOL_TO_BYTE(SCA06_5.OUT))		); Logger.s1:=CONCAT(Logger.s1,';');
Logger.s1:=CONCAT(Logger.s1,BYTE_TO_STRING(BOOL_TO_BYTE(SCA06_6.OUT))		); Logger.s1:=CONCAT(Logger.s1,';');
Logger.s1:=CONCAT(Logger.s1,BYTE_TO_STRING(BOOL_TO_BYTE(SCA06_7.OUT))		); Logger.s1:=CONCAT(Logger.s1,';');
Logger.s1:=CONCAT(Logger.s1,BYTE_TO_STRING(BOOL_TO_BYTE(SCA06_8.OUT))		); Logger.s1:=CONCAT(Logger.s1,';');
Logger.s1:=CONCAT(Logger.s1,BYTE_TO_STRING(BOOL_TO_BYTE(SCA06_9.OUT))		); Logger.s1:=CONCAT(Logger.s1,';');
Logger.s1:=CONCAT(Logger.s1,BYTE_TO_STRING(BOOL_TO_BYTE(SCA06_10.OUT))		); Logger.s1:=CONCAT(Logger.s1,';');
Logger.s1:=CONCAT(Logger.s1,BYTE_TO_STRING(BOOL_TO_BYTE(SCA06_11.OUT))		); Logger.s1:=CONCAT(Logger.s1,';');
Logger.s1:=CONCAT(Logger.s1,BYTE_TO_STRING(BOOL_TO_BYTE(SCA06_12.OUT))		); Logger.s1:=CONCAT(Logger.s1,';');

Logger.s1:=CONCAT(Logger.s1,BYTE_TO_STRING(BOOL_TO_BYTE(SCA06_15.OUT))		); Logger.s1:=CONCAT(Logger.s1,';');
Logger.s1:=CONCAT(Logger.s1,BYTE_TO_STRING(BOOL_TO_BYTE(SCA06_16.OUT))		); Logger.s1:=CONCAT(Logger.s1,';');
(*
Logger.s1:=CONCAT(Logger.s1,BYTE_TO_STRING(BOOL_TO_BYTE(SCA06_17.OUT))		); Logger.s1:=CONCAT(Logger.s1,';');
Logger.s1:=CONCAT(Logger.s1,BYTE_TO_STRING(BOOL_TO_BYTE(SCA06_18.OUT))		); Logger.s1:=CONCAT(Logger.s1,';');
*)
Logger.s1:=CONCAT(Logger.s1,BYTE_TO_STRING(BOOL_TO_BYTE(SCA06_19.OUT))		); Logger.s1:=CONCAT(Logger.s1,';');
Logger.s1:=CONCAT(Logger.s1,BYTE_TO_STRING(BOOL_TO_BYTE(SCA06_20.OUT))		); Logger.s1:=CONCAT(Logger.s1,';');
Logger.s1:=CONCAT(Logger.s1,BYTE_TO_STRING(BOOL_TO_BYTE(SCA06_21.OUT))		); Logger.s1:=CONCAT(Logger.s1,';');
Logger.s1:=CONCAT(Logger.s1,BYTE_TO_STRING(BOOL_TO_BYTE(SCA06_22.OUT))		);


ADDSTRING(ADR(Logger.TData), ADR(Logger.s1), Logger.TLen);
END_ACTION

(* POU Utils Functions/FLT_TAP, ST *)
FUNCTION_BLOCK FLT_TAP
VAR_INPUT
	IN		: BOOL;
	TAP		: BYTE:=4;
	INITEV	: BOOL:=TRUE;
END_VAR
VAR_OUTPUT
	OUT		: BOOL;
	EVH		: BOOL;
	EVL		: BOOL;
END_VAR
VAR
	init	: BOOL:=FALSE;
	cnt		: BYTE;
END_VAR
EVH:=FALSE;
EVL:=FALSE;

IF NOT init THEN
	init := TRUE;
	IF INITEV THEN
		OUT  := NOT IN;
		cnt  := TAP;
	ELSE
		OUT  := IN;
	END_IF
END_IF

IF OUT<>IN THEN
	cnt:=cnt+1;
	IF cnt>TAP THEN
		OUT:=IN;
		cnt:=0;
		IF OUT THEN EVH:=TRUE; ELSE EVL:=TRUE; END_IF
	END_IF
ELSE
	cnt:=0;
END_IF
END_FUNCTION_BLOCK

(* POU TCP_Logger/LogEv, ST *)
FUNCTION LogEv : BOOL
VAR_INPUT
	Level	: en_Logger_ErrLev;
	Object  : en_SYS_Objects;
	Index	: WORD;
	Error	: WORD;
	Message : STRING;
END_VAR
VAR
	s1 : STRING(160);
	i  : INT;
END_VAR
(* Execute error level operations *)
CASE Level OF
	EL_Wrn: 		Sys.Warning:=TRUE;
	EL_Alarm: 		Sys.Alarm  :=TRUE;
	EL_AlarmStop: 	Sys.Alarm  :=TRUE; (* GO TO STOP STATE!! *)
END_CASE

(* Fill lastlog list *)
s1:=CONCAT(Sys.Time_LogString,';Lev=');
s1:=CONCAT(s1,INT_TO_STRING(Level));
s1:=CONCAT(s1,';Obj=');
s1:=CONCAT(s1,INT_TO_STRING(Object));
s1:=CONCAT(s1,';Idx=');
s1:=CONCAT(s1,WORD_TO_STRING(Index));
s1:=CONCAT(s1,';Err=');
s1:=CONCAT(s1,WORD_TO_STRING(Error));
Sys.LastLogs_Dat[Sys.LastLogs_Idx]:=s1;
Sys.LastLogs_Msg[Sys.LastLogs_Idx]:=Message;
Sys.LastLogs_Idx:=Sys.LastLogs_Idx+1;
IF Sys.LastLogs_Idx>5 THEN Sys.LastLogs_Idx:=0; END_IF

(*---------------------------------------------------------------*)
	Logger_Head();
(*---------------------------------------------------------------*)

(* Insert ERR *)
s1:=CONCAT('&ERR=',INT_TO_STRING(Level));
s1:=CONCAT(s1,';');
s1:=CONCAT(s1,INT_TO_STRING(Object));
s1:=CONCAT(s1,';');
s1:=CONCAT(s1,WORD_TO_STRING(Index));
s1:=CONCAT(s1,';');
s1:=CONCAT(s1,WORD_TO_STRING(Error));
s1:=CONCAT(s1,';');
ADDSTRING(ADR(Logger.TData), ADR(s1), Logger.TLen);
s1:=Message;
STR_NOSPACES(ADR(s1));
ADDSTRING(ADR(Logger.TData), ADR(s1), Logger.TLen);

(*---------------------------------------------------------------*)
	Logger_Send();
(*---------------------------------------------------------------*)
END_FUNCTION

(* POU TCP_Logger/Logger_Head, ST *)
FUNCTION Logger_Head : BOOL
VAR
	s1 : STRING(160);
	i  : BYTE;
	dataConvertita: STRING;

END_VAR
Logger.TLen:=0;
(* Set GET header *)
ADDSTRING(ADR(Logger.TData), ADR(Logger_GETSTART), Logger.TLen);

(* Insert Header *)
s1:=INSERT('ID=&V=1&D=',DWORD_TO_STRING(Plant_SN),3);

(* Registrazione nuovo formato dell'ora *)

 s1:=CONCAT(s1,Sys.Time_LogString);
(*
dataConvertita:=REPLACE(Sys.Time_LogString,'T',1,11);
dataConvertita:=CONCAT(dataConvertita,'.000');
dataConvertita:=CONCAT(dataConvertita,SEL(OraLegale,'+01:00','+02:00'));
s1:=CONCAT(s1,dataConvertita);
*)

s1:=CONCAT(s1,'&S=');
IF Sys.Alarm THEN i:=2; ELSIF Sys.Warning THEN i:=1; ELSE i:=0; END_IF
s1:=CONCAT(s1,BYTE_TO_STRING(i));
ADDSTRING(ADR(Logger.TData), ADR(s1), Logger.TLen);
END_FUNCTION

(* POU Utils Functions/ADDSTRING, ST *)
FUNCTION ADDSTRING : BOOL (* Append string to a byte buffer *)
VAR_INPUT
	pTxData: POINTER TO BYTE;
	pString: POINTER TO BYTE;
END_VAR
VAR_IN_OUT
	TxLen: DINT;
END_VAR
VAR
END_VAR
pTxData:=pTxData+TxLen;
WHILE pString^<>0 DO
	pTxData^:=pString^;
	pString:=pString+1;
	pTxData:=pTxData+1;
	TxLen:=TxLen+1;
END_WHILE
END_FUNCTION

(* POU Utils Functions/STR_NOSPACES, ST *)
FUNCTION STR_NOSPACES : BOOL (* Replace spaces and bad chars with allowed ones, used as HTTP-GET validator *)
VAR_INPUT
	pString: POINTER TO BYTE;
END_VAR
VAR
END_VAR
WHILE pString^<>0 DO
	IF pString^=16#20 (* space *) THEN pString^:=16#5F; (*'_'*) END_IF
	pString:=pString+1;
END_WHILE
END_FUNCTION

(* POU TCP_Logger/Logger_Send, ST *)
FUNCTION Logger_Send : BOOL
VAR
	hFile: 	DWORD;
	pos:	DWORD;
END_VAR
(* Finalize string *)
ADDSTRING(ADR(Logger.TData), ADR(Logger_GETEND), Logger.TLen);

(* Read log position *)
pos:=SysFileGetSize(Logger_DataFile);
(* Check log size, bckup and erase if no pending messages *)
IF pos>100000000 (*100M*) THEN
	hFile:=SysFileOpen(Logger_IndexFile,'r');
	IF hFile=0 THEN
		SysFileDelete(Logger_DataFileOld);
		SysFileRename(Logger_DataFile,Logger_DataFileOld);
		pos:=0;
	ELSE
		SysFileClose(hFile);
	END_IF
END_IF
(* Write message on log file *)
hFile:=SysFileOpen(Logger_DataFile,'a');
IF hFile<>0 THEN
	SysFileWrite(hFile, ADR(Logger.TData), Logger.TLen);
	SysFileClose(hFile);
ELSE
	Sys.Warning:=TRUE;
END_IF


(* Check logger status *)
IF Logger.SendReq=FALSE THEN
	(* Set log position for recovery *)
	Logger.SendIdx:=pos;
	(* Copy message data *)
	MEMCPY(ADR(Logger.TData),ADR(Logger.SendData),DINT_TO_WORD(Logger.TLen));
	Logger.SendLen:=Logger.TLen;
	(* Trigger request *)
	Logger.SendReq:=TRUE;
ELSE
	(* Add message position+size in recovery indexes *)
	hFile:=SysFileOpen(Logger_IndexFile,'a');
	SysFileWrite(hFile, ADR(pos), SIZEOF(pos));
	SysFileWrite(hFile, ADR(Logger.TLen), SIZEOF(Logger.TLen));
	SysFileClose(hFile);
END_IF
END_FUNCTION

(* POU Utils Functions/MEMCPY, ST *)
FUNCTION MEMCPY:BOOL
VAR_INPUT
	pSourceAddress:POINTER TO ARRAY[1..2] OF BYTE;
	pDestinationAddress:POINTER TO ARRAY[1..2] OF BYTE;
	BytesToCopy:WORD;
END_VAR
VAR
END_VAR
WHILE (BytesToCopy > 0) DO
	pDestinationAddress^[1]:=pSourceAddress^[1]; (* copy bytes from source to destination *)
	pDestinationAddress:=ADR(pDestinationAddress^[2]); (* increment destination *)
	pSourceAddress:=ADR(pSourceAddress^[2]);(* increment source *)
	BytesToCopy:=BytesToCopy -1; (* decrement number of bytes to copy *)
END_WHILE
END_FUNCTION

(* POU TCP_Logger/Logger_Proc, ST *)
PROGRAM Logger_Proc
VAR
	c1:         	TCPCLIENT;

	Open:	    	BOOL;
	IpAddr:			DWORD;
	InetAddr:		DWORD;
	Connected:  	BOOL;
	Error:      	DINT;
	TxTrig:     	BOOL;
	RxData:			ARRAY [0..MAX_RECEIVE_TCP_CLIENT] OF BYTE;
	RxLen:			DINT;

	Retry:			BYTE;	(* Counter for connection retries *)
	Recovered:		BYTE;	(* Counter for recovered unsent messages *)

	i:				DINT;
	pos:			DWORD;
	hFile:			DWORD;

END_VAR
(*=== State machine ===*)
CASE Logger.Status OF

	S_Logger_UNKNOWN:
		(* Startup *)
		Logger.SendReq:=FALSE;
		Open:=FALSE;
		Logger.Status:=S_Logger_IDLE;

	S_Logger_IDLE:
		(* Wait request *)
		IF Logger.SendReq THEN
			(* Resolve server name or use static IP *)
			IF LEN(Logger_SERVER)=0 THEN
				InetAddr:=SysSockInetAddr(Logger_IP);
			ELSE
				IpAddr:=SysSockGetHostByName(ADR(Logger_SERVER));
				DWORDSWAP(pIn:=ADR(IpAddr), pOut:=ADR(InetAddr));
			END_IF
			TxTrig:=FALSE;
			RxLen:=0;
			(* Open connection *)
			Open:=TRUE;
			Logger.Status:=S_Logger_WAITCONN;
		END_IF

	S_Logger_WAITCONN:
		(* Wait connection *)
		IF Connected THEN
			(* Send data *)
			TxTrig:=TRUE;
			Logger.Status:=S_Logger_WAITTX;
		END_IF
		IF Error>0 THEN
			Open:=FALSE;
			Logger.Status:=S_Logger_ERROR;
		END_IF

	S_Logger_WAITTX:
		(* Wait transmission *)
		IF NOT TxTrig THEN
			Logger.Status:=S_Logger_WAITRESP;
		END_IF
		IF Error>0 THEN
			Open:=FALSE;
			Logger.Status:=S_Logger_ERROR;
		END_IF

	S_Logger_WAITRESP:
		(* Wait response *)
		IF Connected=FALSE (* OR TIMEOUT!! *) THEN
			Open:=FALSE;
			(* Check response *)
			IF RxLen>=4 AND CHKSTRING(pString:=ADR(RxData), pPattern:=ADR(Logger_CHECK)) THEN
				Logger.SendReq:=FALSE;
				Retry:=0;
				(* Check unsent messages to flush *)
				IF Recovered<Logger_RecoverMsgs THEN
					MsgChk();
					IF Logger.SendReq=TRUE THEN
						Recovered:=Recovered+1;
					ELSE
						Recovered:=0;
					END_IF
				ELSE
					Recovered:=0;
				END_IF
				Logger.Status:=S_Logger_IDLE;
			ELSE
				Logger.Status:=S_Logger_ERROR;
			END_IF
		END_IF

	S_Logger_ERROR:
		(* Connection error or send failure *)
		Retry:=Retry+1;
		IF Retry>Logger_ConnRetries THEN
			(* Save message as unsent *)
			MsgSave();
			Logger.SendReq:=FALSE;
			Retry:=0;
		END_IF
		Logger.Status:=S_Logger_IDLE;

ELSE
	Logger.Status:=S_Logger_UNKNOWN;
END_CASE


(*=== Execute client lib ===*)
c1(
	xOpenConnection			:= Open,
	dwInetAddr 				:= InetAddr,
	wPortNumber				:= Logger_PORT,
	ptSendData				:= ADR(Logger.SendData),
	diSendCount				:= Logger.SendLen,
	tConnectWatchdogTime	:= t#10s,
	xStartSend				:= TxTrig,
	aReceiveBuffer			:= RxData,
	diReceiveCount			:= RxLen,
	xConnected				=> Connected,
	diError					=> Error
);

(*=== Process Rx data ===*)
(*IF RxLen>0 THEN
	RxLen:=0;
END_IF*)
END_PROGRAM
ACTION MsgChk:
(* Open index file *)
hFile:=SysFileOpen(Logger_IndexFile,'r');
IF hFile=0 THEN
	RETURN;
END_IF
(* Search oldest message to recover *)
SysFileSetPos(hFile,Logger.LastIdxPos);
Logger.SendLen:=0;
REPEAT
	SysFileRead(hFile, ADR(Logger.SendIdx), SIZEOF(Logger.SendIdx));
	pos:=SysFileGetPos(hFile);
	SysFileRead(hFile, ADR(Logger.SendLen), SIZEOF(Logger.SendLen));
UNTIL
	SysFileEOF(hFile) OR Logger.SendLen<>0
END_REPEAT
SysFileClose(hFile);
(* Delete index file when all messages are recovered *)
IF Logger.SendLen=0 THEN
	Logger.LastIdxPos:=0;
	SysFileDelete(Logger_IndexFile);
	RETURN;
END_IF
(* Recover message data *)
hFile:=SysFileOpen(Logger_DataFile,'r');
IF hFile<>0 THEN
	SysFileSetPos(hFile,Logger.SendIdx);
	SysFileRead(hFile,ADR(Logger.SendData),Logger.SendLen);
	Logger.SendReq:=TRUE;
	SysFileClose(hFile);
END_IF
(* Clear index entry *)
hFile:=SysFileOpen(Logger_IndexFile,'a');
IF hFile<>0 THEN
	SysFileSetPos(hFile,pos);
	i:=0;
	SysFileWrite(hFile, ADR(i), 4);
	Logger.LastIdxPos:=SysFileGetPos(hFile);
	SysFileClose(hFile);
END_IF
END_ACTION
ACTION MsgSave:
(* Add log position in recovery indexes *)
hFile:=SysFileOpen(Logger_IndexFile,'a');
SysFileWrite(hFile, ADR(Logger.SendIdx), SIZEOF(Logger.SendIdx));
SysFileWrite(hFile, ADR(Logger.SendLen), SIZEOF(Logger.SendLen));
SysFileClose(hFile);
END_ACTION

(* POU Utils Functions/TCPCLIENT, ST *)
FUNCTION_BLOCK TCPCLIENT
(***********************************************************************************************************	*)
(* Version: 1.3b                        			          													*)
(* Date: 28.10.2014                   				          							            			*)
(***********************************************************************************************************	*)
(* WAGO Kontakttechnik GmbH Hansastr. 27 32423 Minden(Westf.)													*)
(* Tel. +0049 571/887-0 Fax. +0049 571/887-0																	*)
(* Author: VB																									*)
(***********************************************************************************************************	*)
(*Description:	A TCP client to read and write data with additional connection watchdog							*)
(*History:																										*)
(*Version 1.3b: 28.10.2014: Use DWORD address for IP (Andrea Ravasio)											*)
(*Version 1.3: 11.02.2011: Changes according to 750-880/881											 			*)
(*Version 1.2: 29.08.2007 Bugfix TCP Client																		*)
(*Version 1.1: 15.01.2007 Changes according to FW11																*)
(*Version 1.0: 09.03.2006 Release																				*)
(***********************************************************************************************************	*)
VAR CONSTANT
	STATE_CREATE     				 : BYTE:= 0;
	STATE_OPEN     					 : BYTE:= 1;
	STATE_IOCTL    					 : BYTE:= 2;
	STATE_CONNECT     				 : BYTE:= 10;
	STATE_TX       					 : BYTE:= 20;
	STATE_RX       					 : BYTE:= 30;
	STATE_CLOSE    					 : BYTE:= 40;
	STATE_ERROR_TRAP			     : BYTE:= 200;
END_VAR

VAR_INPUT
	xOpenConnection					: BOOL;
	dwInetAddr						: DWORD; (* <== Use SysSockInetAddr() value or
													swapped bytes order of SysSockGetHostByName() value *)
	wPortNumber						: WORD;
	ptSendData						: POINTER TO ARRAY[0..MAX_SEND_TCP_CLIENT] OF BYTE;
	diSendCount						: DINT;
	tConnectWatchdogTime		    : TIME := t#10s;
END_VAR
VAR_OUTPUT
	xConnected						: BOOL;
	diError 						: DINT := 0;
END_VAR
(* ErrorCodes -----------------------------------------
	16#8001 => No socket descriptor available 
	16#8002 => SysSockSend returns -1 
	16#8003 => Socket was "gracefully closed" 
	16#8004 => switching to none blocking mode fails
	16#8005 => SysSockClose() returns FALSE 
    16#8006 => SysSockConnect() fails
    16#8007 => SysSockSend() fails
	16#8008 => error state machine 
	16#8009 => timeout while waiting for data from server 
------------------------------------------------------------*)
VAR_IN_OUT
	xStartSend							: BOOL;
	aReceiveBuffer						: ARRAY [0..MAX_RECEIVE_TCP_CLIENT] OF BYTE;
	diReceiveCount						: DINT;
END_VAR
VAR
	m_State								: BYTE := 0;
	m_ReceiveBuffer						: ARRAY [0..MAX_RECEIVE_TCP_CLIENT_SOCKET] OF BYTE;
	m_Socket							: DINT;
	m_AddressInfo						: SOCKADDRESS;
	m_BytesReceived						: DINT;
	m_diReturn							: DINT;
	m_xReturn							: BOOL;
	m_IoCtlParameter  					: DINT := 1; (* IOCTL-Parameter for non-blocking mode of sockets *)
	i									: INT;
	T_Connect							: TON;
	m_count								: DINT;
	diOption							: DINT := 1;
	m_Blocking   						: DINT := 0;
END_VAR
IF xOpenConnection THEN
	(* State maschine *)
	CASE  m_State OF

	(* -------------------------------------------------------------------------*)
	STATE_CREATE:
			(* create socket descriptor*)
			m_Socket := SysSockCreate(diAddressFamily	:= SOCKET_AF_INET,
													 diType		:= SOCKET_STREAM,
													 diProtocol := SOCKET_IPPROTO_TCP);
			IF m_Socket >= 0 THEN
			(*Set Push-Bit*)
				IF ADR(%MW0)=16#30000000  OR ADR(%MW0)=16#20000000 THEN (*841 or 881*)
					SysSockSetOption(
						diSocket:=m_Socket,
						diLevel:=6,
						diOption:=SOCKET_TCP_NODELAY,
						pOptionValue:=ADR(diOption),
						diOptionLength:=SIZEOF(diOption));
				ELSE
						;
				END_IF
				m_State := STATE_IOCTL; (* succesful *)
			ELSE
				diError := 16#8001;  (* no socket descriptor available *)
				m_State := STATE_ERROR_TRAP;
			END_IF

	(* -------------------------------------------------------------------------*)
	STATE_IOCTL: (* change  socket mode  to none blocking *)
		m_diReturn := SysSockIoctl( m_Socket, SOCKET_FIONBIO, ADR(m_IoCtlParameter));
		IF m_diReturn <> 0 THEN
			m_AddressInfo.sin_family := SOCKET_AF_INET;
			m_AddressInfo.sin_port := SysSockNtohs(wPortNumber);
			m_AddressInfo.sin_addr := dwInetAddr;
			m_State := STATE_CONNECT;
		ELSE
			diError := 16#8004;  (* switching to none blocking mode fails *)
			m_State := STATE_ERROR_TRAP;
		END_IF


	(* -------------------------------------------------------------------------*)
	STATE_CONNECT: (* connect with server *)
		T_Connect(IN:=TRUE , PT:=tConnectWatchdogTime);(*activate watchdog for establishing connection to a server*)
		m_xReturn := SysSockConnect ( m_Socket, ADR(m_AddressInfo),  SIZEOF(m_AddressInfo));
		IF m_xReturn THEN (* succesful *)
			IF xStartSend THEN
				m_State := STATE_TX;(*transmit data*)
			ELSE
				m_State := STATE_RX;(*wait for data from server*)
			END_IF
			xConnected:=TRUE;
			T_Connect(IN:=FALSE);
		ELSE
			IF T_Connect.Q THEN
				diError := 16#8006;  (* connect fails *)
				xConnected:=FALSE;
				T_Connect(IN:=FALSE);
				m_State := STATE_ERROR_TRAP;
				SysSockClose( m_Socket);
			ELSE
				m_State := STATE_CONNECT;(*client still  tries to set up connection*)
			END_IF
		END_IF


	STATE_TX:	 (* send TCP-message *)
		m_diReturn := SysSockSend(diSocket := m_Socket,
								  pbyBuffer := ADR(ptSendData^[0]),
								  diBufferSize := diSendCount-m_count,
								  diFlags := 0);

		CASE m_diReturn OF
		-1:	(* ERROR *)
			T_Connect(IN:=TRUE , PT:=CONNECT_WATCHDOG_TIME);(*activate watchdog to check communication*)
			IF t_Connect.Q THEN
				diError := 16#8007;
				T_Connect(IN:=FALSE);
				m_State:=STATE_CLOSE;
			END_IF
		0: (* socket was "gracefully closed" *)
			m_State := STATE_CLOSE;
			diError := 16#8003;
		ELSE (* succesful *)
			m_count:=m_count+m_diReturn;
			IF m_count>=diSendCount THEN
				diError := 16#0000;
				m_State := STATE_RX;
				m_count:=0;
				xStartSend:=FALSE;
			END_IF
			T_Connect(IN:=FALSE);
		END_CASE

	(* -------------------------------------------------------------------------*)
	STATE_RX: (* process receive data *)
			m_BytesReceived := SysSockRecv(	diSocket 	:= m_Socket,
										pbyBuffer 	:= ADR(m_ReceiveBuffer),		(* Address of receive buffer *)
										diBufferSize:= SIZEOF(m_ReceiveBuffer),
										diFlags		:= 0);

			CASE m_BytesReceived OF
			-1:	(* No data available or error occured *)
				T_Connect(IN:=TRUE , PT:=tConnectWatchdogTime);(*activate watchdog to check communication*)
				IF t_Connect.Q THEN
					diError:=16#8009;
					T_Connect(IN:=FALSE);
					m_State:=STATE_CLOSE;
				END_IF
				IF xStartSend THEN
					m_State:=STATE_TX	;(* WAIT IN THIS STATE  and check for arriving data or new send command*)
				END_IF;
			0: (* socket was "gracefully closed"  *)
				m_State:=STATE_CLOSE;
				diError := 16#8003;
			ELSE (* succesful *)
				diError := 16#0000;
				T_Connect(IN:=FALSE);
				(* Copy received data into receive buffer *)
				FOR i:= 0 TO DINT_TO_INT(m_BytesReceived	)-1 DO
					aReceiveBuffer[diReceiveCount]:= m_ReceiveBuffer[i];
					diReceiveCount:=(diReceiveCount+1) MOD SIZEOF(aReceiveBuffer);
				END_FOR

			END_CASE

	(* -------------------------------------------------------------------------*)
	STATE_CLOSE : (* close socket *)
		IF ADR(%MW0)=16#30000000  OR ADR(%MW0)=16#20000000 THEN (*841 or 881*)
			;
		ELSE
			SysSockShutdown(m_Socket, 0);;(*870*)
		END_IF
		m_xReturn := SysSockClose( m_Socket);
		m_Socket := -1;
		m_State := 0; (* succesful *)
		xConnected:=FALSE;
		T_Connect(IN:=FALSE);
	(* -------------------------------------------------------------------------*)
	STATE_ERROR_TRAP: (* error handling *)
		xConnected:=FALSE;

	ELSE  (* Bad FSM code trap  *)
			m_State:= STATE_ERROR_TRAP;
			diError:= 16#8008;
	END_CASE

ELSE(*close connection*)
	IF m_Socket >= 0 THEN
		IF ADR(%MW0)=16#30000000  OR ADR(%MW0)=16#20000000 THEN (*841 or 881*)
			;
		ELSE
			SysSockShutdown(m_Socket, 0);;(*870*)
		END_IF
		SysSockClose( m_Socket);
	END_IF
	m_Socket := -1;
	diError := 16#0000;
	m_State := STATE_CREATE;
	xConnected:=FALSE;
	T_Connect(IN:=FALSE);
END_IF
END_FUNCTION_BLOCK

(* POU Utils Functions/DWORDSWAP, ST *)
FUNCTION DWORDSWAP:BOOL
VAR_INPUT
	pIn:POINTER TO ARRAY[1..4] OF BYTE;
	pOut:POINTER TO ARRAY[1..4] OF BYTE;
END_VAR
VAR
END_VAR
pOut^[1]:=pIn^[4];
pOut^[2]:=pIn^[3];
pOut^[3]:=pIn^[2];
pOut^[4]:=pIn^[1];
END_FUNCTION

(* POU Utils Functions/CHKSTRING, ST *)
FUNCTION CHKSTRING : BOOL
VAR_INPUT
	pString: POINTER TO BYTE;
	pPattern: POINTER TO BYTE;
END_VAR
VAR
END_VAR
CHKSTRING:=TRUE;
WHILE pPattern^<>0 AND CHKSTRING DO
	IF pPattern^<>pString^ THEN CHKSTRING:=FALSE; END_IF
	pString:=pString+1;
	pPattern:=pPattern+1;
END_WHILE
END_FUNCTION

(* POU TCP_Remote/Remote_Proc, ST *)
PROGRAM Remote_Proc
VAR
	s1:         	TCPSERVER;
	Enable: 		BOOL;
	Connected: 		BOOL;
	Error: 			DINT;

	TxData:			ARRAY [0..MAX_SEND_TCP_SERVER] OF BYTE;
	TxLen:			DINT;
	TxTrig:			BOOL;

	RxData:			ARRAY [0..MAX_RECEIVE_TCP_SERVER] OF BYTE;
	RxLen:			DINT;

	Status:			DINT;

	(* Command interpreter *)

	Cmd_Buf:		ARRAY [0..MAX_RECEIVE_TCP_SERVER] OF BYTE;
	Cmd_Buf_U16:	POINTER TO WORD;
	Cmd_Buf_INT:	POINTER TO INT;
	Cmd_BufLen:		WORD;
	Cmd_St:			WORD;

	Cmd_Obj:		WORD;
	Cmd_ObjIdx:		WORD;
	Cmd_C:			WORD;
	Cmd_R:			WORD;
	Cmd_CLen:		WORD;
	Cmd_RLen:		WORD;

	i : WORD;
	j : INT;

	moreno: DT;

		(* per aggiornare la data e l'ora *)
	SetAnno: INT;
	SetMese: INT;
	SetGiorno: INT;
	SetOra: INT;
	SetMinuti: INT;
	SetSecondi: INT;



END_VAR
(*=== State machine ===*)
CASE Status OF
	0: (* Startup *)
		TxLen:=0; TxTrig:=FALSE;
		RxLen:=0;
		Enable:=TRUE;
		Status:=1;

	1: (* Wait incoming connection *)
		IF Connected THEN
			(* Log access *)
			LogEv(EL_Log,EO_VPN,1,5,'Remote');
			(* Send welcome message *)
			(*ADDSTRING(pTxData:=ADR(TxData), pString:=ADR(Remote_WELCOME), TxLen:=TxLen);
			TxTrig:=TRUE;*)
			Cmd_BufLen:=0;
			Cmd_St:=0;
			Status:=2;
		END_IF
		IF Error>1 THEN
			Enable:=FALSE;
			Status:=0;
		END_IF

	2: (* Wait command *)
		IF RxLen>0 THEN
			(*=== Interpreter start ===*)
			IF Cmd_BufLen+(RxLen/2)>=MAX_RECEIVE_TCP_SERVER THEN
				(* ERROR *)
				Cmd_BufLen:=0;
			ELSE
				i:=HEXTORAW(pString:=ADR(RxData), StringLen:=DINT_TO_WORD(RxLen), pData:=ADR(Cmd_Buf[Cmd_BufLen]));
				Cmd_BufLen:=Cmd_BufLen+i;
			END_IF
			IF Cmd_BufLen>=8 THEN
				Cmd_Buf_U16:=ADR(Cmd_Buf[6]);
				IF Cmd_BufLen>=(8+Cmd_Buf_U16^) THEN
					Cmd_CLen:=Cmd_Buf_U16^;
					Cmd_Buf_U16:=ADR(Cmd_Buf[0]); Cmd_Obj:=Cmd_Buf_U16^;
					Cmd_Buf_U16:=ADR(Cmd_Buf[2]); Cmd_ObjIdx:=Cmd_Buf_U16^;
					Cmd_Buf_U16:=ADR(Cmd_Buf[4]); Cmd_C:=Cmd_Buf_U16^;
					Command();
					Cmd_BufLen:=0;
				END_IF
			END_IF
			(*=== Interpreter end ===*)
			RxLen:=0;
		END_IF
		IF NOT Connected THEN
			Status:=0;
		END_IF

ELSE
	Status:=0;
END_CASE


(*=== Execute server lib ===*)
s1(
	xEnable				:= Enable,
	wPortNumber			:= Remote_PORT,
	tServerTimeOut		:= t#15m,
	ptSendData			:= ADR(TxData),
	diSendCount			:= TxLen,
	xStartSend			:= TxTrig,
	aReceiveBuffer		:= RxData,
	diReceiveCount		:= RxLen,
	xClientConnected	=> Connected,
	diError				=> Error
);
END_PROGRAM
ACTION cmd_CAL:
(* Check index *)
IF Cmd_ObjIdx<2 OR Cmd_ObjIdx>3 THEN
	Cmd_R:=2;
	RETURN;
END_IF

(* Process command *)
CASE Cmd_C OF

	1: (* GET CLIMATIC *)
		Cmd_RLen:=20;
		FOR i:=0 TO 4 DO
			CASE Cmd_ObjIdx OF
				2:	j:=DINT_TO_INT(CAL02_Clima.Points[i].X);
				3:	j:=DINT_TO_INT(CAL03_Clima.Points[i].X);
			END_CASE
				TxLen:=TxLen+RAWTOHEX(ADR(j),2,ADR(TxData[TxLen]));

			CASE Cmd_ObjIdx OF
				2: j:=DINT_TO_INT(CAL02_Clima.Points[i].Y);
				3: j:=DINT_TO_INT(CAL03_Clima.Points[i].Y);
			END_CASE
				TxLen:=TxLen+RAWTOHEX(ADR(j),2,ADR(TxData[TxLen]));
			END_FOR

	2: (* SET CLIMATIC *)
		IF Cmd_CLen<>20 THEN
			Cmd_R:=4;
		ELSE
			CASE Cmd_ObjIdx OF
				2:
				FOR i:=0 TO 4 DO
					Cmd_Buf_INT:=ADR(Cmd_Buf[8+4*i]); j:=Cmd_Buf_INT^;
					CAL02_Clima.Points[i].X:=INT_TO_DINT(j);
					Cmd_Buf_INT:=ADR(Cmd_Buf[10+4*i]); j:=Cmd_Buf_INT^;
					CAL02_Clima.Points[i].Y:=INT_TO_DINT(j);
				END_FOR
				3:
				FOR i:=0 TO 4 DO
					Cmd_Buf_INT:=ADR(Cmd_Buf[8+4*i]); j:=Cmd_Buf_INT^;
					CAL03_Clima.Points[i].X:=INT_TO_DINT(j);
					Cmd_Buf_INT:=ADR(Cmd_Buf[10+4*i]); j:=Cmd_Buf_INT^;
					CAL03_Clima.Points[i].Y:=INT_TO_DINT(j);
				END_FOR
			END_CASE



		END_IF

	3: (* Reset Caldia *)

		CASE Cmd_ObjIdx OF

			2:	CAL02.TCP_ResetCAL:=TRUE;
			3:	CAL03.TCP_ResetCAL:=TRUE;

		END_CASE

	4: (* SET Tempi delay On Off Ccaldaia  *)
		CASE Cmd_ObjIdx OF
			2:	Cmd_Buf_U16:=ADR(Cmd_Buf[8]);
				CAL02.OnDelay := DWORD_TO_TIME((Cmd_Buf_U16^)*60*1000); 			(* Delay ON*)
				Cmd_Buf_U16:=ADR(Cmd_Buf[10]);
				CAL02.OffDelay := DWORD_TO_TIME((Cmd_Buf_U16^)*60*1000);			(* Delay OFF *)
			3:	Cmd_Buf_U16:=ADR(Cmd_Buf[8]);
				CAL03.OnDelay := DWORD_TO_TIME((Cmd_Buf_U16^)*60*1000);				(* Delay ON*)
				Cmd_Buf_U16:=ADR(Cmd_Buf[10]);
				CAL03.OffDelay := DWORD_TO_TIME((Cmd_Buf_U16^)*60*1000);			(* Delay OFF *)

		END_CASE


	5: (* GET Tempi delay On Off Caldaia *)
		Cmd_RLen:=4;

			CASE Cmd_ObjIdx OF

			2:	j:=DWORD_TO_WORD(TIME_TO_DWORD((CAL02.OnDelay)/60/1000));
				TxLen:=TxLen+RAWTOHEX(ADR(j),2,ADR(TxData[TxLen]));
				j:=DWORD_TO_WORD(TIME_TO_DWORD((CAL02.OffDelay)/60/1000));
				TxLen:=TxLen+RAWTOHEX(ADR(j),2,ADR(TxData[TxLen]));
			3: 	j:=DWORD_TO_WORD(TIME_TO_DWORD((CAL03.OnDelay)/60/1000));
				TxLen:=TxLen+RAWTOHEX(ADR(j),2,ADR(TxData[TxLen]));
				j:=DWORD_TO_WORD(TIME_TO_DWORD((CAL03.OffDelay)/60/1000));
				TxLen:=TxLen+RAWTOHEX(ADR(j),2,ADR(TxData[TxLen]));

		END_CASE









ELSE
	Cmd_R:=3;
END_CASE
END_ACTION
ACTION cmd_CIRD:
IF Cmd_ObjIdx<1 OR Cmd_ObjIdx>6 THEN
	Cmd_R:=2;
	RETURN;
END_IF

(* Process command *)
CASE Cmd_C OF

	1:	(* Force CIR On *)
		CASE Cmd_ObjIdx OF

			1:	CIRD01.CIR_RUN_REQ := TRUE;
				CIRD01.CIR_STOP_REQ := FALSE;
			2:	CIRD02.CIR_RUN_REQ := TRUE;
				CIRD02.CIR_STOP_REQ := FALSE;

		END_CASE

	2:	(* Force CIR Off *)
		CASE Cmd_ObjIdx OF

			1:	CIRD01.CIR_STOP_REQ := TRUE;
				CIRD01.CIR_RUN_REQ	:= FALSE;
			2:	CIRD02.CIR_STOP_REQ := TRUE;
				CIRD02.CIR_RUN_REQ	:= FALSE;

		END_CASE

	3:	(* Release force *)
		CASE Cmd_ObjIdx OF

			1:	CIRD01.CIR_RUN_REQ	:= FALSE;
				CIRD01.CIR_STOP_REQ := FALSE;
			2:	CIRD02.CIR_RUN_REQ	:= FALSE;
				CIRD02.CIR_STOP_REQ := FALSE;
		END_CASE


	4: (* SET Tempi delay On Off Circolatori  *)
		CASE Cmd_ObjIdx OF
			1:	Cmd_Buf_U16:=ADR(Cmd_Buf[8]);
				CIRD01.OnDelay := DWORD_TO_TIME((Cmd_Buf_U16^)*60*1000); 			(* Delay ON*)
				Cmd_Buf_U16:=ADR(Cmd_Buf[10]);
				CIRD01.OffDelay := DWORD_TO_TIME((Cmd_Buf_U16^)*60*1000);			(* Delay OFF *)
			2:	Cmd_Buf_U16:=ADR(Cmd_Buf[8]);
				CIRD02.OnDelay := DWORD_TO_TIME((Cmd_Buf_U16^)*60*1000);				(* Delay ON*)
				Cmd_Buf_U16:=ADR(Cmd_Buf[10]);
				CIRD02.OffDelay := DWORD_TO_TIME((Cmd_Buf_U16^)*60*1000);			(* Delay OFF *)

		END_CASE


	5: (* GET Tempi delay On Off Circolatori *)
		Cmd_RLen:=4;
			CASE Cmd_ObjIdx OF

			1:	j:=DWORD_TO_WORD(TIME_TO_DWORD((CIRD01.OnDelay)/60/1000));
				TxLen:=TxLen+RAWTOHEX(ADR(j),2,ADR(TxData[TxLen]));
				j:=DWORD_TO_WORD(TIME_TO_DWORD((CIRD01.OffDelay)/60/1000));
				TxLen:=TxLen+RAWTOHEX(ADR(j),2,ADR(TxData[TxLen]));
			2: 	j:=DWORD_TO_WORD(TIME_TO_DWORD((CIRD02.OnDelay)/60/1000));
				TxLen:=TxLen+RAWTOHEX(ADR(j),2,ADR(TxData[TxLen]));
				j:=DWORD_TO_WORD(TIME_TO_DWORD((CIRD02.OffDelay)/60/1000));
				TxLen:=TxLen+RAWTOHEX(ADR(j),2,ADR(TxData[TxLen]));

		END_CASE

	6: (* SET Modalità di Funzionamento *)
		CASE Cmd_ObjIdx OF
			1:	Cmd_Buf_U16:=ADR(Cmd_Buf[8]);
				CIRD01.mode := WORD_TO_BYTE(Cmd_Buf_U16^); 										(* Modalità di Funzionamento *)
			2:	Cmd_Buf_U16:=ADR(Cmd_Buf[8]);
				CIRD02.mode := WORD_TO_BYTE(Cmd_Buf_U16^); 										(* Modalità di Funzionamento *)

		END_CASE
ELSE
	Cmd_R:=3;
END_CASE
END_ACTION
ACTION Cmd_CRON:
(* Check index *)
IF Cmd_ObjIdx<1 OR Cmd_ObjIdx>4 THEN
	Cmd_R:=2;
	RETURN;
END_IF

(* Process command *)
CASE Cmd_C OF

	1: (* GET PROFILE *)
		IF Cmd_CLen<>3 THEN
			Cmd_R:=4;
		ELSE
			(* Load profile *)
			CronEd.CN_Sel:=WORD_TO_BYTE(Cmd_ObjIdx);
			Cmd_Buf_U16:=ADR(Cmd_Buf[8]);
			CronEd.CN_YSel:=Cmd_Buf_U16^;
			IF Cmd_Buf[10]<=10 THEN
				CronEd.PR_Sel:=Cmd_Buf[10];
				CronEd.PR_Load_Exe();
				(* Response data *)
				Cmd_RLen:=192;
				TxLen:=TxLen+RAWTOHEX(ADR(CronEd.PR.Setpoint),192,ADR(TxData[TxLen]));
			ELSE
				Cmd_R:=6;
			END_IF
		END_IF

	2: (* SET PROFILE *)
		IF Cmd_CLen<>(3+192) THEN
			Cmd_R:=4;
		ELSE
			(* Save profile *)
			CronEd.CN_Sel:=WORD_TO_BYTE(Cmd_ObjIdx);
			Cmd_Buf_U16:=ADR(Cmd_Buf[8]);
			CronEd.CN_YSel:=Cmd_Buf_U16^;
			IF Cmd_Buf[10]<=10 THEN
				CronEd.PR_Sel:=Cmd_Buf[10];
				MEMCPY(ADR(Cmd_Buf[11]),ADR(CronEd.PR.Setpoint),192);
				CronEd.PR_Save_Exe();
			ELSE
				Cmd_R:=6;
			END_IF
		END_IF

	5: (* GET CALENDAR MONTH *)
		IF Cmd_CLen<>3 THEN
			Cmd_R:=4;
		ELSE
			(* Load calendar *)
			CronEd.CN_Sel:=WORD_TO_BYTE(Cmd_ObjIdx);
			Cmd_Buf_U16:=ADR(Cmd_Buf[8]);
			CronEd.CN_YSel:=Cmd_Buf_U16^;
			IF Cmd_Buf[10]>=1 AND Cmd_Buf[10]<=12 THEN
				CronEd.CA_Sel:=Cmd_Buf[10];
				CronEd.CA_Load_Exe();
				(* Response data *)
				Cmd_RLen:=32;
				TxLen:=TxLen+RAWTOHEX(ADR(CronEd.CA.Profile),32,ADR(TxData[TxLen]));
			ELSE
				Cmd_R:=6;
			END_IF
		END_IF

	6: (* SET CALENDAR MONTH *)
		IF Cmd_CLen<>(3+32) THEN
			Cmd_R:=4;
		ELSE
			(* Save calendar *)
			CronEd.CN_Sel:=WORD_TO_BYTE(Cmd_ObjIdx);
			Cmd_Buf_U16:=ADR(Cmd_Buf[8]);
			CronEd.CN_YSel:=Cmd_Buf_U16^;
			IF Cmd_Buf[10]>=1 AND Cmd_Buf[10]<=12 THEN
				CronEd.CA_Sel:=Cmd_Buf[10];
				MEMCPY(ADR(Cmd_Buf[11]),ADR(CronEd.CA.Profile),32);
				CronEd.CA_Save_Exe();
			ELSE
				Cmd_R:=6;
			END_IF
		END_IF

	9: (* CRON RESTART *)
		CASE Cmd_ObjIdx OF
			(*1: CRON01.InitOK:=FALSE;*)
			1: THER01.InitOK:=FALSE;
			2: THER02.InitOK:=FALSE;
			3: THER03.InitOK:=FALSE;
			4: THER04.InitOK:=FALSE;

		END_CASE

	10: (* SET Isteresi  *)
		CASE Cmd_ObjIdx OF
			1:	Cmd_Buf_U16:=ADR(Cmd_Buf[8]);
				THER01.Histeresys := Cmd_Buf_U16^; 			(* Isteresi*)
			2:	Cmd_Buf_U16:=ADR(Cmd_Buf[8]);
				THER02.Histeresys := Cmd_Buf_U16^; 			(* Isteresi*)
			3:	Cmd_Buf_U16:=ADR(Cmd_Buf[8]);
				THER03.Histeresys := Cmd_Buf_U16^; 			(* Isteresi*)
			4:	Cmd_Buf_U16:=ADR(Cmd_Buf[8]);
				THER04.Histeresys := Cmd_Buf_U16^; 			(* Isteresi*)
		END_CASE

	11: (* GET isteresi *)
		Cmd_RLen:=2;
		CASE Cmd_ObjIdx OF


			1: j:=(THER01.Histeresys);
				TxLen:=TxLen+RAWTOHEX(ADR(j),2,ADR(TxData[TxLen]));
			2: j:=(THER02.Histeresys);
				TxLen:=TxLen+RAWTOHEX(ADR(j),2,ADR(TxData[TxLen]));
			3: j:=(THER03.Histeresys);
				TxLen:=TxLen+RAWTOHEX(ADR(j),2,ADR(TxData[TxLen]));
			4: j:=(THER04.Histeresys);
				TxLen:=TxLen+RAWTOHEX(ADR(j),2,ADR(TxData[TxLen]));

		END_CASE

ELSE
	Cmd_R:=3;
END_CASE
END_ACTION
ACTION Cmd_CTB:
(* Check index *)
IF Cmd_ObjIdx<>1 THEN
	Cmd_R:=2;
	RETURN;
END_IF

(* Process command *)
CASE Cmd_C OF

	1: (* START REFRESH *)
		CTBSCAN01.Refresh:=TRUE;
	2: (* START REFRESH *)
		CTBSCAN01.Refresh:=FALSE;
	3: (* START RESCAN/SEARCH *)
		CTBSCAN01.Rescan:=TRUE;
	4: (* STOP  RESCAN/SEARCH *)
		CTBSCAN01.Rescan:=FALSE;

ELSE
	Cmd_R:=3;
END_CASE
END_ACTION
ACTION cmd_EV:
IF Cmd_ObjIdx<1 OR Cmd_ObjIdx>3 THEN
	Cmd_R:=2;
	RETURN;
END_IF

(* Process command *)
CASE Cmd_C OF

	1:	(* Force CIR On *)
		CASE Cmd_ObjIdx OF

			2:	EV02.EV_OPEN_REQ := TRUE;
				EV02.EV_CLOSE_REQ := FALSE;
			3:	EV03.EV_OPEN_REQ := TRUE;
				EV03.EV_CLOSE_REQ := FALSE;
		END_CASE

	2:	(* Force CIR Off *)
		CASE Cmd_ObjIdx OF

			2:	EV02.EV_CLOSE_REQ := TRUE;
				EV02.EV_OPEN_REQ	:= FALSE;
			3:	EV03.EV_CLOSE_REQ := TRUE;
				EV03.EV_OPEN_REQ	:= FALSE;
		END_CASE

	3:	(* Release force *)
		CASE Cmd_ObjIdx OF

			2:	EV02.EV_OPEN_REQ	:= FALSE;
				EV02.EV_CLOSE_REQ := FALSE;
			3:	EV03.EV_OPEN_REQ	:= FALSE;
				EV03.EV_CLOSE_REQ := FALSE;
		END_CASE


	4: (* SET Tempi delay On Off   *)
		CASE Cmd_ObjIdx OF
			2:	Cmd_Buf_U16:=ADR(Cmd_Buf[8]);
				EV02.OnDelay := DWORD_TO_TIME((Cmd_Buf_U16^)*60*1000); 			(* Delay ON*)
				Cmd_Buf_U16:=ADR(Cmd_Buf[10]);
				EV02.OffDelay := DWORD_TO_TIME((Cmd_Buf_U16^)*60*1000);			(* Delay OFF *)
			3:	Cmd_Buf_U16:=ADR(Cmd_Buf[8]);
				EV03.OnDelay := DWORD_TO_TIME((Cmd_Buf_U16^)*60*1000);				(* Delay ON*)
				Cmd_Buf_U16:=ADR(Cmd_Buf[10]);
				EV03.OffDelay := DWORD_TO_TIME((Cmd_Buf_U16^)*60*1000);			(* Delay OFF *)
		END_CASE


	5: (* GET Tempi delay On Off  *)
		Cmd_RLen:=4;
			CASE Cmd_ObjIdx OF

			2:	j:=DWORD_TO_WORD(TIME_TO_DWORD((EV02.OnDelay)/60/1000));
				TxLen:=TxLen+RAWTOHEX(ADR(j),2,ADR(TxData[TxLen]));
				j:=DWORD_TO_WORD(TIME_TO_DWORD((EV02.OffDelay)/60/1000));
				TxLen:=TxLen+RAWTOHEX(ADR(j),2,ADR(TxData[TxLen]));
			3: 	j:=DWORD_TO_WORD(TIME_TO_DWORD((EV03.OnDelay)/60/1000));
				TxLen:=TxLen+RAWTOHEX(ADR(j),2,ADR(TxData[TxLen]));
				j:=DWORD_TO_WORD(TIME_TO_DWORD((EV03.OffDelay)/60/1000));
				TxLen:=TxLen+RAWTOHEX(ADR(j),2,ADR(TxData[TxLen]));
		END_CASE


ELSE
	Cmd_R:=3;
END_CASE
END_ACTION
ACTION cmd_GAS:
IF Cmd_ObjIdx<1 OR Cmd_ObjIdx>2 THEN
	Cmd_R:=2;
	RETURN;
END_IF

(* Process command *)
CASE Cmd_C OF

(*

	1: (* GET Offset impostato *)
		Cmd_RLen:=4;
			CASE Cmd_ObjIdx OF
			1:	j:=Dint_to_int(Conteggio_GAS1.Conteggio_GAS1)/65535);
				TxLen:=TxLen+RAWTOHEX(ADR(j),2,ADR(TxData[TxLen]));
				j:=Dint_to_int((Conteggio_GAS1.Conteggio_GAS1)/65535-(Conteggio_GAS1.Conteggio_GAS1)/65535));
				TxLen:=TxLen+RAWTOHEX(ADR(j),2,ADR(TxData[TxLen]));
			2:	j:=Dint_to_int(Conteggio_GAS2.Conteggio_GAS2)/65535);
				TxLen:=TxLen+RAWTOHEX(ADR(j),2,ADR(TxData[TxLen]));
				j:=Dint_to_int((Conteggio_GAS2.Conteggio_GAS2)/65535-(Conteggio_GAS2.Conteggio_GAS2)/65535));
				TxLen:=TxLen+RAWTOHEX(ADR(j),2,ADR(TxData[TxLen]));


		END_CASE

*)



	2:	(* Comando Offset Contatori GAS *)
		CASE Cmd_ObjIdx OF

		(**** il dato in ricezione è in 2 word quindi deve essere costruito il valore corretto ***)
		(**** per questo impianto la soluzione migliore è questa , va rivisto il bloccheto GAS ***)


		1: (* Scrittura Limite accettabile di pedite *)
			Cmd_Buf_U16:=ADR(Cmd_Buf[8]);
			OffsetContatoreGAS1_1W:= Cmd_Buf_U16^;
			Cmd_Buf_U16:=ADR(Cmd_Buf[10]);
			OffsetContatoreGAS1_2W:= Cmd_Buf_U16^;

			OffsetGAS1:=OffsetContatoreGAS1_2W *65536 + OffsetContatoreGAS1_1W;
			ChangeGAS1:=TRUE;

			ConteggioGAS1.Offset();


		2: (* Scrittura Limite accettabile di pedite *)
			Cmd_Buf_U16:=ADR(Cmd_Buf[8]);
			OffsetContatoreGAS2_1W:= Cmd_Buf_U16^;
			Cmd_Buf_U16:=ADR(Cmd_Buf[10]);
			OffsetContatoreGAS2_2W:= Cmd_Buf_U16^;

			OffsetGAS2:=OffsetContatoreGAS2_2W *65536 + OffsetContatoreGAS2_1W;
			ChangeGAS2:=TRUE;
			ConteggioGAS2.Offset();

		END_CASE

ELSE
	Cmd_R:=3;
END_CASE
END_ACTION
ACTION Cmd_SYS:
(* Check index *)
IF Cmd_ObjIdx<>0 THEN
	Cmd_R:=2;
	RETURN;
END_IF

(* Process command *)
CASE Cmd_C OF

	0: (* ECHO *)
		IF Cmd_CLen<>0 THEN
			TxLen:=0;
		END_IF

	1: (* LOG REQUEST *)
		LogTrig();

	2: (* REARM *)
		Sys.Warning:=FALSE;
		Sys.Alarm:=FALSE;
		Sys.AlarmStop:=FALSE;

	3: (* GET INFO1 *)
		Cmd_RLen:=6;
		TxLen:=TxLen+RAWTOHEX(ADR(Plant_SN),4,ADR(TxData[TxLen]));
		TxLen:=TxLen+RAWTOHEX(ADR(Plant_SW_VER),2,ADR(TxData[TxLen]));


	4: (*  Scrivo i Parametri gestione Impianto   *)

			Cmd_Buf_U16:=ADR(Cmd_Buf[8]);
			DelayAllarmeTemperaturaNonRaggiunta := Cmd_Buf_U16^; 			(* Ritardo Allarme dall'avvio Caldaia*)
			Cmd_Buf_U16:=ADR(Cmd_Buf[10]);
			DeltaInterventoAllarmeTempeaturaNonRaggiuta := Cmd_Buf_U16^;	(* Delta Soglia Temperatura per Allarme Temperatura Non Raggiunta *)
			Cmd_Buf_U16:=ADR(Cmd_Buf[12]);
			OffsetSetPointManuale := Cmd_Buf_U16^; 					(* Offest Perdite Scambiatore  *)

	5: (*  Leggi i parametri gestione Impianto  *)

			Cmd_RLen:=14;
			j:=(DelayAllarmeTemperaturaNonRaggiunta);   				(* Ritardo Allarme dall'avvio Caldaia*)
			TxLen:=TxLen+RAWTOHEX(ADR(j),2,ADR(TxData[TxLen]));
			j:=(DeltaInterventoAllarmeTempeaturaNonRaggiuta);			(* Delta Soglia Temperatura per Allarme Temperatura Non Raggiunta *)
			TxLen:=TxLen+RAWTOHEX(ADR(j),2,ADR(TxData[TxLen]));
			j:=(OffsetSetPointManuale);									(* Offest Perdite Scambiatore  *)
			TxLen:=TxLen+RAWTOHEX(ADR(j),2,ADR(TxData[TxLen]));

(*	6: (*  Scrivo i Parametri gestione Impianto - Antigelo   *)

			Cmd_Buf_U16:=ADR(Cmd_Buf[8]);
			SogliaMinStartAntigelo := Cmd_Buf_U16^; 			(* Soglia mininma Start Antigelo *)
			Cmd_Buf_U16:=ADR(Cmd_Buf[10]);
			SogliaMinStopAntigelo := Cmd_Buf_U16^;				(* Soglia Massima Stop Antigelo *)
			Cmd_Buf_U16:=ADR(Cmd_Buf[12]);
			BitAbilitaAntigelo :=INT_TO_BOOL( Cmd_Buf_U16^); 	(* Abilitazione Antigelo  *)

	7: (*  Leggi i parametri gestione Impianto - Antigelo *)

			Cmd_RLen:=14;
			j:=(SogliaMinStartAntigelo); 							(* Soglia mininma Start Antigelo *)
			TxLen:=TxLen+RAWTOHEX(ADR(j),2,ADR(TxData[TxLen]));
			j:=(SogliaMinStopAntigelo);								(* Soglia Massima Stop Antigelo *)
			TxLen:=TxLen+RAWTOHEX(ADR(j),2,ADR(TxData[TxLen]));
			j:=BOOL_TO_INT(BitAbilitaAntigelo);						(* Abilitazione Antigelo  *)
			TxLen:=TxLen+RAWTOHEX(ADR(j),2,ADR(TxData[TxLen]));

	10: (*  Scrivo i Parametri per la gestione della velocità dei circolatori sui primari   *)

			Cmd_Buf_U16:=ADR(Cmd_Buf[8]);
			PercVelMin := Cmd_Buf_U16^;
			Cmd_Buf_U16:=ADR(Cmd_Buf[10]);
			PercVelMax := Cmd_Buf_U16^;
			Cmd_Buf_U16:=ADR(Cmd_Buf[12]);
			ErroreTempMax := Cmd_Buf_U16^;
			Cmd_Buf_U16:=ADR(Cmd_Buf[14]);
			ErroreTempMin := Cmd_Buf_U16^;

	11: (*  Leggo i Parametri per la gestione della velocità dei circolatori sui primari   *)

			Cmd_RLen:=8;
			j:=(PercVelMin);
			TxLen:=TxLen+RAWTOHEX(ADR(j),2,ADR(TxData[TxLen]));
			j:=(PercVelMax);
			TxLen:=TxLen+RAWTOHEX(ADR(j),2,ADR(TxData[TxLen]));
			j:=(ErroreTempMax);
			TxLen:=TxLen+RAWTOHEX(ADR(j),2,ADR(TxData[TxLen]));
			j:=(ErroreTempMin);
			TxLen:=TxLen+RAWTOHEX(ADR(j),2,ADR(TxData[TxLen]));


	12: (*  Scrivo i Parametri per la gestione della velocità dei circolatori sui primari   *)


				Cmd_Buf_U16:=ADR(Cmd_Buf[8]);
				CAS01.DeltaTempThr := Cmd_Buf_U16^;
				Cmd_Buf_U16:=ADR(Cmd_Buf[10]);
				CAS01.Tmonitor_Off := DWORD_TO_TIME((Cmd_Buf_U16^)*60*1000);
				Cmd_Buf_U16:=ADR(Cmd_Buf[12]);
				CAS01.Tmonitor_On := DWORD_TO_TIME((Cmd_Buf_U16^)*60*1000);

	13: (*  Leggo i Parametri per la gestione della velocità dei circolatori sui primari   *)


				Cmd_RLen:=6;
				j:=(CAS01.DeltaTempThr);
				TxLen:=TxLen+RAWTOHEX(ADR(j),2,ADR(TxData[TxLen]));
				j:=DWORD_TO_WORD(TIME_TO_DWORD((CAS01.Tmonitor_Off)/60/1000));
				TxLen:=TxLen+RAWTOHEX(ADR(j),2,ADR(TxData[TxLen]));
				j:=DWORD_TO_WORD(TIME_TO_DWORD((CAS01.Tmonitor_On)/60/1000));
				TxLen:=TxLen+RAWTOHEX(ADR(j),2,ADR(TxData[TxLen]));


*)


	14: (*  Imposto data e ora del PLC  *)


			Cmd_Buf_U16:=ADR(Cmd_Buf[8]);
			SetAnno:= Cmd_Buf_U16^; 												(* Anno *)
			Cmd_Buf_U16:=ADR(Cmd_Buf[10]);
			SetMese:= Cmd_Buf_U16^;												 	(* mese *)
			Cmd_Buf_U16:=ADR(Cmd_Buf[12]);
			SetGiorno:=( Cmd_Buf_U16^);											 	(* Giorno *)
			Cmd_Buf_U16:=ADR(Cmd_Buf[14]);
			SetOra:=( Cmd_Buf_U16^); 												(* ora *)
			Cmd_Buf_U16:=ADR(Cmd_Buf[16]);
			SetMinuti:= ( Cmd_Buf_U16^);										 	(* Minuti *)
			Cmd_Buf_U16:=ADR(Cmd_Buf[18]);
			SetSecondi:= ( Cmd_Buf_U16^);										 	(* secondi *)

	(*		SysRtcSetTime(SetDataTime(DWORD_TO_INT(ADR(Cmd_Buf[8])),				(* Anno *)
										DWORD_TO_INT(ADR(Cmd_Buf[10])),				(* mese *)
										DWORD_TO_INT(ADR(Cmd_Buf[11])),				(* Giorno *)
										DWORD_TO_INT(ADR(Cmd_Buf[12])),				(* ora *)
										DWORD_TO_INT(ADR(Cmd_Buf[13])),				(* Minuti *)
										DWORD_TO_INT(ADR(Cmd_Buf[14]))				(* secondi *)
										)); *)

		SysRtcSetTime((SetDataTime(SetAnno,SetMese,SetGiorno,SetOra,SetMinuti,SetSecondi)));


ELSE
	Cmd_R:=3;
END_CASE
END_ACTION
ACTION Command:
(* Default response OK/NODATA *)
Cmd_R:=0;
Cmd_RLen:=0;
TxLen:=16;

(* Check object *)
CASE Cmd_Obj OF

	EO_SYS:
		Cmd_SYS();

	EO_CTB:
		Cmd_CTB();

	EO_CIRD:
		Cmd_CIRD();

	EO_EV:
		Cmd_EV();

	EO_CRON:
		Cmd_CRON();

	EO_CAL:
		Cmd_CAL();

	EO_GAS:
		Cmd_GAS();

ELSE
	Cmd_R:=1;
END_CASE

(* Generate response *)
IF TxLen>0 THEN
	RAWTOHEX(ADR(Cmd_Obj)	,2,ADR(TxData[ 0]));
	RAWTOHEX(ADR(Cmd_ObjIdx),2,ADR(TxData[ 4]));
	RAWTOHEX(ADR(Cmd_R)		,2,ADR(TxData[ 8]));
	RAWTOHEX(ADR(Cmd_RLen)	,2,ADR(TxData[12]));
	TxTrig:=TRUE;
END_IF
END_ACTION

(* POU Utils Functions/TCPSERVER, ST *)
FUNCTION_BLOCK TCPSERVER
(***********************************************************************************************************	*)
(* Version: 1.6                                    			          											*)
(* Date: 11.02.2011                                   					          							    *)
(***********************************************************************************************************	*)
(* WAGO Kontakttechnik GmbH Hansastr. 27 32423 Minden(Westf.)													*)
(* Tel. +0049 571/887-0 Fax. +0049 571/887-0																	*)
(* Author: VB																									*)
(***********************************************************************************************************	*)
(*Description:	A TCP server to read and write data													       		*)
(*Historie:																										*)
(*Version 1.6: 11.02.2011: Changes according to 750-880/881											 			*)
(*Version 1.5: 27.11.2008 Bugfix allow reuse port																*)
(*Version 1.4: 13.10.2008 Bugfix transmitting large data														*)
(*Version 1.3: 15.01.2007 Changes according to FW11																*)
(*Version 1.2: 09.03.2006 Changes for socket handle 0											       			*)
(*Version 1.1: 14.02.2005 Release																				*)
(***********************************************************************************************************	*)
VAR CONSTANT
	STATE_INIT     				 : BYTE:= 0;
	STATE_OPEN     				 : BYTE:= 1;
	STATE_TX       				 : BYTE:= 20;
	STATE_RX       				 : BYTE:= 30;
	STATE_CLOSE    				 : BYTE:= 40;
	STATE_ERROR_TRAP		 	 : BYTE:= 200;
END_VAR
VAR_INPUT
	xEnable    					: BOOL;	 (* Set TRUE to enable function block *)
	wPortNumber					: WORD;  (* Port *)
	tServerTimeOut				: TIME:=t#50s;
	ptSendData					: POINTER TO ARRAY[0..MAX_SEND_TCP_SERVER] OF BYTE;
	diSendCount					: DINT;
END_VAR
VAR_OUTPUT
	xClientConnected  			: BOOL:= FALSE;
	diError 					: DINT:= 0;
END_VAR
(* Status Codes -----------------------------------------
	16#8001 => No socket descriptor available 
	16#8002 => SysSockBind fails 
	16#8003 => SysSockListen fails 
	16#8004 => switching to none blocking mode fails
	16#8005 => SysSockClose() returns FALSE 
    16#8006 => SysSockConnect() fails
    16#8007 => SysSockSend() fails
	16#8008 => error state machine 
	16#8009 => timeout while waiting for data from server 
	16#0001 => server waiting for client to establish connection
------------------------------------------------------------*)
VAR_IN_OUT
	xStartSend					: BOOL;
	aReceiveBuffer				: ARRAY [0..MAX_RECEIVE_TCP_SERVER] OF BYTE;
	diReceiveCount				: DINT;
END_VAR

VAR
	m_State    					: BYTE:= 0;
	m_ReceiveBuffer				: ARRAY [0..MAX_RECEIVE_TCP_SERVER_SOCKET] OF BYTE;
	m_ServerSocket				: DINT:= SOCKET_INVALID;
	m_Socket					: DINT:= SOCKET_INVALID;
	m_AddressInfo				: SOCKADDRESS;
	m_BytesReceived				: DINT;
	m_diReturn					: DINT;
	m_xReturn					: BOOL;
	m_SizeSockadr				: DWORD;
	m_ConnectionWatchdog		: TON;
	m_Flags						: DINT;
	m_NoneBlocking   			: DINT:= 1;
	m_Blocking   				: DINT:= 0;
	i							: INT;
	m_count						: DINT;
	diOption					: DINT := 1;
	on: DINT;
END_VAR
IF xEnable THEN
	CASE m_State OF
		STATE_INIT:
			(* Create Socket *)
			m_ServerSocket:= SysSockCreate( SOCKET_AF_INET, SOCKET_STREAM, 0);
			IF m_ServerSocket = SOCKET_INVALID THEN
				(* *)
				diError:= 16#8001;
				m_State:= STATE_ERROR_TRAP;
				RETURN;
			ELSE
				;
			END_IF
			(* Address bindings *)
			(********************)
			on:=1;
			SysSockSetOption( m_ServerSocket, SOCKET_SOL, SOCKET_SO_REUSEADDR, ADR(on), SIZEOF(on) );

			m_AddressInfo.sin_family:= SOCKET_AF_INET;
			m_AddressInfo.sin_port  := SysSockHtons( wPortNumber);
			m_AddressInfo.sin_addr  := SOCKET_INADDR_ANY;
			IF NOT SysSockBind( m_ServerSocket, ADR(m_AddressInfo), SIZEOF(m_AddressInfo)) THEN
				diError:= 16#8002;
				m_State:= STATE_ERROR_TRAP;
				RETURN;
			END_IF
			(* Wait for connections *)
			(************************)
			IF NOT SysSockListen( m_ServerSocket, 1) THEN
				diError:= 16#8003;
				m_State:= STATE_ERROR_TRAP;
			END_IF

			(* Puts SOCKET in NonBlocking mode *)
			m_diReturn:= SysSockIoctl( m_ServerSocket, SOCKET_FIONBIO, ADR(m_NoneBlocking));

			m_State:= STATE_OPEN;


